REGION Network 5: DataIn - Sollevatori
   RUNG wire#powerrail
      "ValveMachine_PB_Connector"(Enable := TRUE, HMI_PB := "A03_HMI".MB3.Button.A0301.P2.Sollevatori, LB_PB_Rest := FALSE, LB_PB_Work := FALSE, LB_PB_StartStop := FALSE, Other_PB := "A03_HMI".MB3.Button.PB_Empty.Valve, PB => "A0301_Fermi_P2".Sollevatori[1].DataIn.PB)
   END_RUNG
   // the same network as SCL:
   "ValveMachine_PB_Connector"(Enable := TRUE,
                           HMI_PB := "A03_HMI".MB3.Button.A0301.P2.Sollevatori,
                           LB_PB_Rest := FALSE,
                           LB_PB_Work := FALSE,
                           LB_PB_StartStop := FALSE,
                           Other_PB := "A03_HMI".MB3.Button.PB_Empty.Valve,
                           PB => "A0301_Fermi_P2".Sollevatori[1].DataIn.PB);
END_REGION

REGION Network 6 (SCL): DataIn - Sollevatori [1..6]
   // TRASFERIMENTO STATO PULSANTI - Comando manuale diretto 
   "A0301_Fermi_P2".Sollevatori[6].DataIn.PB := "A0301_Fermi_P2".Sollevatori[5].DataIn.PB := "A0301_Fermi_P2".Sollevatori[4].DataIn.PB :=
   "A0301_Fermi_P2".Sollevatori[3].DataIn.PB := "A0301_Fermi_P2".Sollevatori[2].DataIn.PB := "A0301_Fermi_P2".Sollevatori[1].DataIn.PB;
END_REGION

REGION Network 7: << RICHIAMO STAZIONE 2 - FERMI P2 >>
   RUNG wire#powerrail
      "A0301_Fermi_P2"(AreaInterface := "Area03".AreaInterface, ZSI := "F_DB".ZSI_Zone21, DSI := "F_DB".DSI_V_Air_A0301_A0302, DataIn :=, CIn :=, Config := "PrjConfig_A03".A0301.Fermi_P2, MachineInterface =>, COut =>)
   END_RUNG
   // the same network as SCL:
   "A0301_Fermi_P2"(AreaInterface := "Area03".AreaInterface,   // "A0301_Fermi_P2_FB"
                    ZSI := "F_DB".ZSI_Zone21,
                    DSI := "F_DB".DSI_V_Air_A0301_A0302,
                    Config := "PrjConfig_A03".A0301.Fermi_P2);
END_REGION

REGION Network 8 (SCL): << TRASFERIMENTO stati DataOut >>
   REGION COMANDO DELLE USCITE FERMI P2

       // Fermi blocco prodotto Stazione P2 - RIPOSO
       // 
       "A0301_CinghiaTrasporto_1.1_V_Rest_7" := "A0301_Fermi_P2".Fermi[1].DataOut.RestSolenoid;
       "A0301_CinghiaTrasporto_2.1_V_Rest_7" := "A0301_Fermi_P2".Fermi[2].DataOut.RestSolenoid;
       "A0301_CinghiaTrasporto_3.1_V_Rest_7" := "A0301_Fermi_P2".Fermi[3].DataOut.RestSolenoid;
       "A0301_CinghiaTrasporto_4.1_V_Rest_7" := "A0301_Fermi_P2".Fermi[4].DataOut.RestSolenoid;
       "A0301_CinghiaTrasporto_5.1_V_Rest_7" := "A0301_Fermi_P2".Fermi[5].DataOut.RestSolenoid;
       "A0301_CinghiaTrasporto_6.1_V_Rest_7" := "A0301_Fermi_P2".Fermi[6].DataOut.RestSolenoid;

       // Fermi blocco prodotto Stazione P2 - LAVORO
       // 
       "A0301_CinghiaTrasporto_1.1_V_Work_8" := "A0301_Fermi_P2".Fermi[1].DataOut.WorkSolenoid;
       "A0301_CinghiaTrasporto_2.1_V_Work_8" := "A0301_Fermi_P2".Fermi[2].DataOut.WorkSolenoid;
       "A0301_CinghiaTrasporto_3.1_V_Work_8" := "A0301_Fermi_P2".Fermi[3].DataOut.WorkSolenoid;
       "A0301_CinghiaTrasporto_4.1_V_Work_8" := "A0301_Fermi_P2".Fermi[4].DataOut.WorkSolenoid;
       "A0301_CinghiaTrasporto_5.1_V_Work_8" := "A0301_Fermi_P2".Fermi[5].DataOut.WorkSolenoid;
       "A0301_CinghiaTrasporto_6.1_V_Work_8" := "A0301_Fermi_P2".Fermi[6].DataOut.WorkSolenoid;
   END_REGION ;

   REGION COMANDO DELLE USCITE SOLLEVATORE P2
       // Sollevatore Semi guscio prodotto Stazione P2 - RIPOSO
       // 
       "A0301_CinghiaTrasporto_1.1_V_Rest_5" := "A0301_Fermi_P2".Sollevatori[1].DataOut.RestSolenoid;
       "A0301_CinghiaTrasporto_2.1_V_Rest_5" := "A0301_Fermi_P2".Sollevatori[2].DataOut.RestSolenoid;
       "A0301_CinghiaTrasporto_3.1_V_Rest_5" := "A0301_Fermi_P2".Sollevatori[3].DataOut.RestSolenoid;
       "A0301_CinghiaTrasporto_4.1_V_Rest_5" := "A0301_Fermi_P2".Sollevatori[4].DataOut.RestSolenoid;
       "A0301_CinghiaTrasporto_5.1_V_Rest_5" := "A0301_Fermi_P2".Sollevatori[5].DataOut.RestSolenoid;
       "A0301_CinghiaTrasporto_6.1_V_Rest_5" := "A0301_Fermi_P2".Sollevatori[6].DataOut.RestSolenoid;

       // Sollevatore Semi guscio prodotto Stazione P2 - LAVORO
       // 
       "A0301_CinghiaTrasporto_1.1_V_Work_6" := "A0301_Fermi_P2".Sollevatori[1].DataOut.WorkSolenoid;
       "A0301_CinghiaTrasporto_2.1_V_Work_6" := "A0301_Fermi_P2".Sollevatori[2].DataOut.WorkSolenoid;
       "A0301_CinghiaTrasporto_3.1_V_Work_6" := "A0301_Fermi_P2".Sollevatori[3].DataOut.WorkSolenoid;
       "A0301_CinghiaTrasporto_4.1_V_Work_6" := "A0301_Fermi_P2".Sollevatori[4].DataOut.WorkSolenoid;
       "A0301_CinghiaTrasporto_5.1_V_Work_6" := "A0301_Fermi_P2".Sollevatori[5].DataOut.WorkSolenoid;
       "A0301_CinghiaTrasporto_6.1_V_Work_6" := "A0301_Fermi_P2".Sollevatori[6].DataOut.WorkSolenoid;

   END_REGION ;*)
END_REGION
END_FUNCTION

FUNCTION_BLOCK "A0301_Fermi_P2_FB"   // FB62, LAD
TITLE = == GESTIONE DELLA STAZIONE P2 ==
// stored: MemoryReserve 100, SetENOAutomatically false
   VAR_INPUT
      AreaInterface : "AreaInterface";
      ZSI : "udt_ZoneSafetyInterface";
      DSI : "udt_DeviceSafetyInterface";
      DataIn : Struct
         OP_Rest_PB : Bool;
         OP_Work_PB : Bool;
      END_STRUCT;
      CIn : Struct
         Manager_Fermi : "ValveMachine_Manager";
         Manager_Sollevatori : "ValveMachine_Manager";
         SemiAut : Bool;
         P1 : Struct
            Fermi : "ValveMachine_COut";
            Pareggiatore : "ValveMachine_COut";
         END_STRUCT;
         Trasporto : "SpeedMachine_COut";
         Sts_Ribalta : Struct
            Pos0_Reached : Bool;
            Pos1_Reached : Bool;
            Pos2_Reached : Bool;
            Pos3_Reached : Bool;
         END_STRUCT;
      END_STRUCT;
      Config : Struct
         Fermi : Array[1..6] of "ValveMachine_Config";
         Sollevatori : Array[1..6] of "ValveMachine_Config";
         DelayMissingCondition : Time := T#3s;
      END_STRUCT;
   END_VAR
   VAR_OUTPUT
      MachineInterface : "MachineInterface";
      COut : Struct
         Fermi : "ValveMachine_COut";
         Sollevatori : "ValveMachine_COut";
      END_STRUCT;
   END_VAR
   VAR
      Alarm : Struct
         Fermi : Array[1..6] of "ValveAlr";
         Sollevatori { S7_SetPoint := 'True'} : Array[1..6] of "ValveAlr";
      END_STRUCT;
      Warning : Struct
         OP_REST_MissingCnd : Bool;   // Mancanza comando arresto
         OP_WORK_MissingCnd : Bool;   // Mancanza consenso lavoro
         Fermi : Array[1..6] of "ValveMachine_Wng";
         Sollevatori { S7_SetPoint := 'True'} : Array[1..6] of "ValveMachine_Wng";
      END_STRUCT;
      HMI : Struct
         Selection : Array[1..6] of Bool;   // 0=Disable / 1=Enable Pin
         FermiSts { S7_SetPoint := 'True'} : "UDT_HMI-Sts_ValvePosA0301";
         SollevatoriSts { S7_SetPoint := 'True'} : "UDT_HMI-Sts_ValvePosA0301";
      END_STRUCT;
      Sts : Struct
         Fermi_AlarmPresence : Bool;
         Sollevatori_AlarmPresence : Bool;
         OP_CanMoveFreely : Bool;
         OP_Rest_Cnd : Bool;
         Op_Work_Cnd : Bool;
      END_STRUCT;
      Ctrl : Struct
         OP_Rest_Man : Bool;
         OP_Work_Man : Bool;
         OP_Rest_Aut : Bool;
         OP_Work_Aut : Bool;
         OP_Rest : Bool;
         OP_Work : Bool;
      END_STRUCT;
      Fermi : Array[1..6] of "ValveMachine_FB";
      Sollevatori { S7_SetPoint := 'True'} : Array[1..6] of "ValveMachine_FB";
      AUX : Struct
         OP_Rest_PB : Bool;
         OP_Work_PB : Bool;
      END_STRUCT;
      TON_OP_REST_MissingCnd { S7_SetPoint := 'True'} : TON_TIME;
      TON_OP_WORK_MissingCnd { S7_SetPoint := 'True'} : TON_TIME;
      TON_Anticipi : Struct
         Rest : Struct
            Sollevatori { S7_SetPoint := 'True'} : IEC_TIMER;
         END_STRUCT;
         Work : Struct
            Sollevatori : IEC_TIMER;
         END_STRUCT;
      END_STRUCT;
   END_VAR
   VAR_TEMP
      PE : Struct
         OP_Rest_PB : Bool;
         OP_Work_PB : Bool;
      END_STRUCT;
      Anticipi : Struct
         Sollevatori : Struct
            COut_Work : Bool;
            COut_Rest : Bool;
            Not_Ls_Work : Bool;
            Not_Ls_Rest : Bool;
         END_STRUCT;
      END_STRUCT;
   END_VAR
   VAR_TEMP   // added for the SCL form of the ladder/FBD networks
      _w1 : Bool;
      _w2 : Bool;
      _w3 : Bool;
      _w4 : Bool;
   END_VAR
BEGIN

REGION Network 2: Anticipi Movimento LAVORO
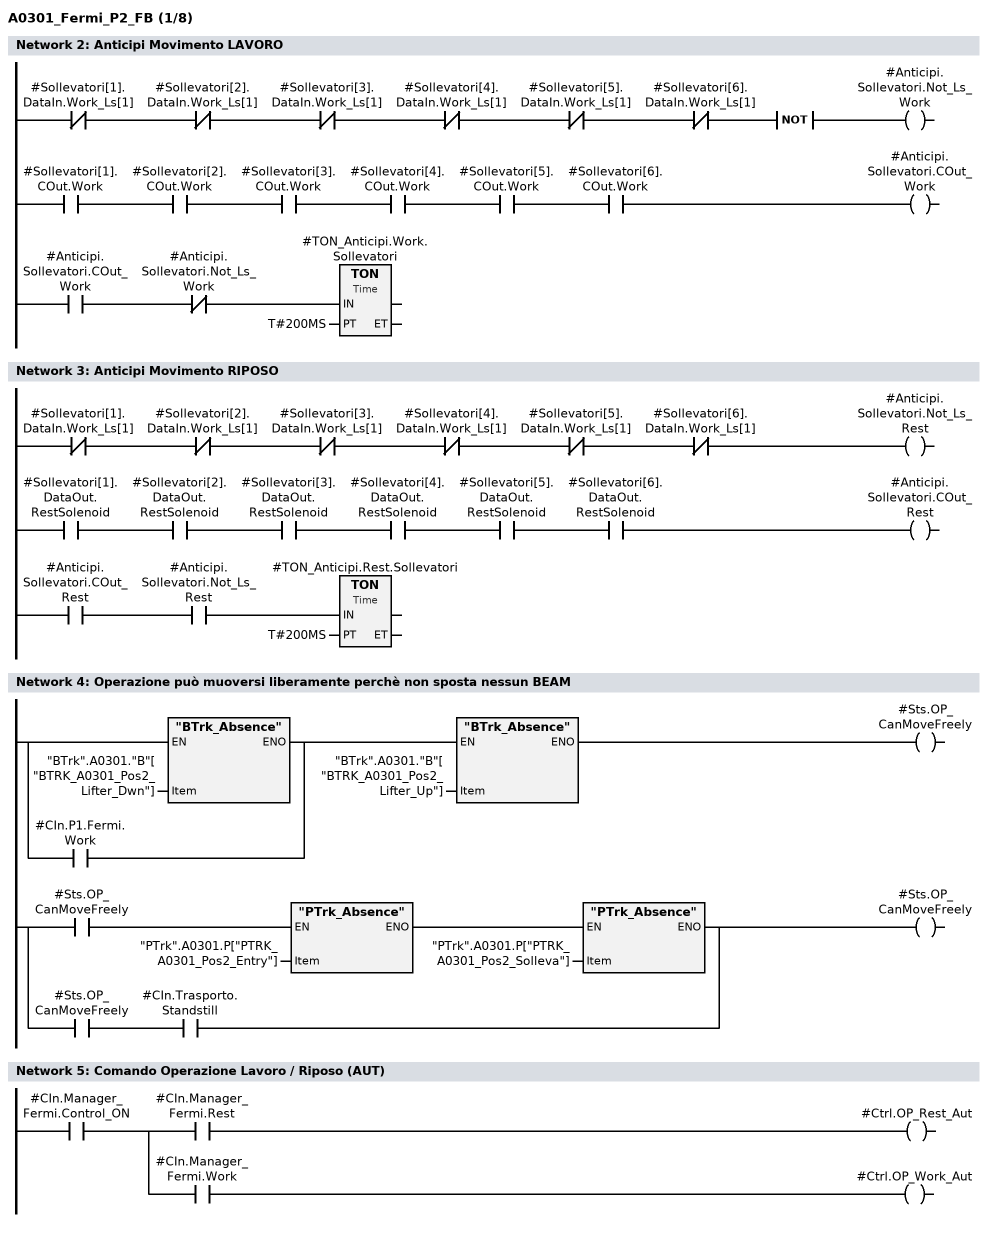
   RUNG wire#powerrail
      I_Contact( #Sollevatori[1].DataIn.Work_Ls[1] )
      I_Contact( #Sollevatori[2].DataIn.Work_Ls[1] )
      I_Contact( #Sollevatori[3].DataIn.Work_Ls[1] )
      I_Contact( #Sollevatori[4].DataIn.Work_Ls[1] )
      I_Contact( #Sollevatori[5].DataIn.Work_Ls[1] )
      I_Contact( #Sollevatori[6].DataIn.Work_Ls[1] )
      Not()
      Coil( #Anticipi.Sollevatori.Not_Ls_Work )
   END_RUNG
   RUNG wire#powerrail
      Contact( #Sollevatori[1].COut.Work )
      Contact( #Sollevatori[2].COut.Work )
      Contact( #Sollevatori[3].COut.Work )
      Contact( #Sollevatori[4].COut.Work )
      Contact( #Sollevatori[5].COut.Work )
      Contact( #Sollevatori[6].COut.Work )
      Coil( #Anticipi.Sollevatori.COut_Work )
   END_RUNG
   RUNG wire#powerrail
      Contact( #Anticipi.Sollevatori.COut_Work )
      I_Contact( #Anticipi.Sollevatori.Not_Ls_Work )
      { S7_Templates := "time_type := Time" } #TON_Anticipi.Work.Sollevatori.TON(pt := T#200MS, et =>)
   END_RUNG
   // the same network as SCL:
   #Anticipi.Sollevatori.Not_Ls_Work := NOT (NOT #Sollevatori[1].DataIn.Work_Ls[1] AND NOT #Sollevatori[2].DataIn.Work_Ls[1] AND NOT #Sollevatori[3].DataIn.Work_Ls[1] AND NOT #Sollevatori[4].DataIn.Work_Ls[1] AND NOT #Sollevatori[5].DataIn.Work_Ls[1] AND NOT #Sollevatori[6].DataIn.Work_Ls[1]);
   #Anticipi.Sollevatori.COut_Work := #Sollevatori[1].COut.Work AND #Sollevatori[2].COut.Work AND #Sollevatori[3].COut.Work AND #Sollevatori[4].COut.Work AND #Sollevatori[5].COut.Work AND #Sollevatori[6].COut.Work;
   #TON_Anticipi.Work.Sollevatori.TON(IN := #Anticipi.Sollevatori.COut_Work AND NOT #Anticipi.Sollevatori.Not_Ls_Work,
                           PT := T#200MS);
END_REGION

REGION Network 3: Anticipi Movimento RIPOSO
   RUNG wire#powerrail
      I_Contact( #Sollevatori[1].DataIn.Work_Ls[1] )
      I_Contact( #Sollevatori[2].DataIn.Work_Ls[1] )
      I_Contact( #Sollevatori[3].DataIn.Work_Ls[1] )
      I_Contact( #Sollevatori[4].DataIn.Work_Ls[1] )
      I_Contact( #Sollevatori[5].DataIn.Work_Ls[1] )
      I_Contact( #Sollevatori[6].DataIn.Work_Ls[1] )
      Coil( #Anticipi.Sollevatori.Not_Ls_Rest )
   END_RUNG
   RUNG wire#powerrail
      Contact( #Sollevatori[1].DataOut.RestSolenoid )
      Contact( #Sollevatori[2].DataOut.RestSolenoid )
      Contact( #Sollevatori[3].DataOut.RestSolenoid )
      Contact( #Sollevatori[4].DataOut.RestSolenoid )
      Contact( #Sollevatori[5].DataOut.RestSolenoid )
      Contact( #Sollevatori[6].DataOut.RestSolenoid )
      Coil( #Anticipi.Sollevatori.COut_Rest )
   END_RUNG
   RUNG wire#powerrail
      Contact( #Anticipi.Sollevatori.COut_Rest )
      Contact( #Anticipi.Sollevatori.Not_Ls_Rest )
      { S7_Templates := "time_type := Time" } #TON_Anticipi.Rest.Sollevatori.TON(pt := T#200MS, et =>)
   END_RUNG
   // the same network as SCL:
   #Anticipi.Sollevatori.Not_Ls_Rest := NOT #Sollevatori[1].DataIn.Work_Ls[1] AND NOT #Sollevatori[2].DataIn.Work_Ls[1] AND NOT #Sollevatori[3].DataIn.Work_Ls[1] AND NOT #Sollevatori[4].DataIn.Work_Ls[1] AND NOT #Sollevatori[5].DataIn.Work_Ls[1] AND NOT #Sollevatori[6].DataIn.Work_Ls[1];
   #Anticipi.Sollevatori.COut_Rest := #Sollevatori[1].DataOut.RestSolenoid AND #Sollevatori[2].DataOut.RestSolenoid AND #Sollevatori[3].DataOut.RestSolenoid AND #Sollevatori[4].DataOut.RestSolenoid AND #Sollevatori[5].DataOut.RestSolenoid AND #Sollevatori[6].DataOut.RestSolenoid;
   #TON_Anticipi.Rest.Sollevatori.TON(IN := #Anticipi.Sollevatori.COut_Rest AND #Anticipi.Sollevatori.Not_Ls_Rest,
                           PT := T#200MS);
END_REGION

REGION Network 4: Operazione può muoversi liberamente perchè non sposta nessun BEAM
   RUNG wire#powerrail
      "BTrk_Absence"(Item := "BTrk".A0301."B"["BTRK_A0301_Pos2_Lifter_Dwn"])
      wire#w1
      "BTrk_Absence"(Item := "BTrk".A0301."B"["BTRK_A0301_Pos2_Lifter_Up"])
      Coil( #Sts.OP_CanMoveFreely )
   END_RUNG
   RUNG wire#powerrail
      Contact( #CIn.P1.Fermi.Work )
   END_RUNG wire#w1
   RUNG wire#powerrail
      Contact( #Sts.OP_CanMoveFreely )
      "PTrk_Absence"(Item := "PTrk".A0301.P["PTRK_A0301_Pos2_Entry"])
      "PTrk_Absence"(Item := "PTrk".A0301.P["PTRK_A0301_Pos2_Solleva"])
      wire#w2
      Coil( #Sts.OP_CanMoveFreely )
   END_RUNG
   RUNG wire#powerrail
      Contact( #Sts.OP_CanMoveFreely )
      Contact( #CIn.Trasporto.Standstill )
   END_RUNG wire#w2
   // the same network as SCL:
   "BTrk_Absence"(Item := "BTrk".A0301."B"["BTRK_A0301_Pos2_Lifter_Dwn"], ENO => #_w1);
   "BTrk_Absence"(EN := #_w1 OR #CIn.P1.Fermi.Work,
                  Item := "BTrk".A0301."B"["BTRK_A0301_Pos2_Lifter_Up"],
                  ENO => #_w2);
   #Sts.OP_CanMoveFreely := #_w2;
   "PTrk_Absence"(EN := #Sts.OP_CanMoveFreely, Item := "PTrk".A0301.P["PTRK_A0301_Pos2_Entry"], ENO => #_w3);
   "PTrk_Absence"(EN := #_w3, Item := "PTrk".A0301.P["PTRK_A0301_Pos2_Solleva"], ENO => #_w4);
   #Sts.OP_CanMoveFreely := #_w4 OR (#Sts.OP_CanMoveFreely AND #CIn.Trasporto.Standstill);
END_REGION

REGION Network 5: Comando Operazione Lavoro / Riposo (AUT)
   RUNG wire#powerrail
      Contact( #CIn.Manager_Fermi.Control_ON )
      wire#w1
      Contact( #CIn.Manager_Fermi.Rest )
      Coil( #Ctrl.OP_Rest_Aut )
   END_RUNG
   RUNG wire#w1
      Contact( #CIn.Manager_Fermi.Work )
      Coil( #Ctrl.OP_Work_Aut )
   END_RUNG
   // the same network as SCL:
   #Ctrl.OP_Rest_Aut := #CIn.Manager_Fermi.Control_ON AND #CIn.Manager_Fermi.Rest;
   #Ctrl.OP_Work_Aut := #CIn.Manager_Fermi.Control_ON AND #CIn.Manager_Fermi.Work;
END_REGION

REGION Network 6: Comando Operazione Lavoro / Riposo (MAN)
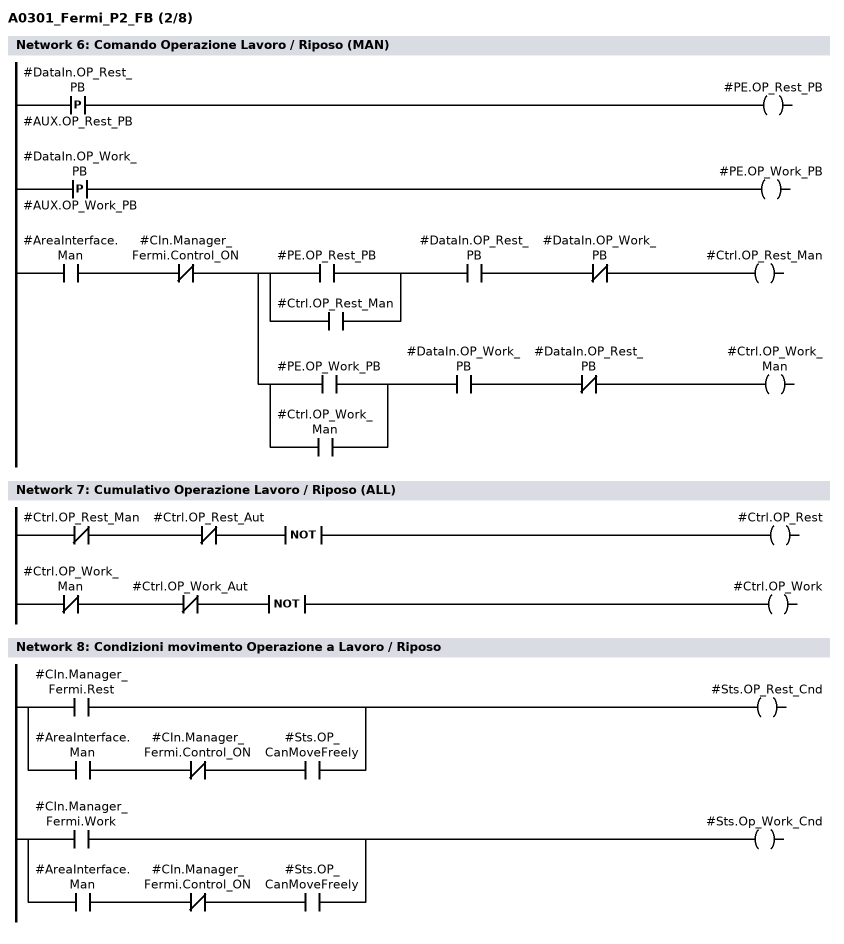
   RUNG wire#powerrail
      P_Contact(operand := #DataIn.OP_Rest_PB, bit := #AUX.OP_Rest_PB)
      Coil( #PE.OP_Rest_PB )
   END_RUNG
   RUNG wire#powerrail
      P_Contact(operand := #DataIn.OP_Work_PB, bit := #AUX.OP_Work_PB)
      Coil( #PE.OP_Work_PB )
   END_RUNG
   RUNG wire#powerrail
      Contact( #AreaInterface.Man )
      I_Contact( #CIn.Manager_Fermi.Control_ON )
      wire#w1
      Contact( #PE.OP_Rest_PB )
      wire#w2
      Contact( #DataIn.OP_Rest_PB )
      I_Contact( #DataIn.OP_Work_PB )
      Coil( #Ctrl.OP_Rest_Man )
   END_RUNG
   RUNG wire#w1
      Contact( #Ctrl.OP_Rest_Man )
   END_RUNG wire#w2
   RUNG wire#w1
      Contact( #PE.OP_Work_PB )
      wire#w3
      Contact( #DataIn.OP_Work_PB )
      I_Contact( #DataIn.OP_Rest_PB )
      Coil( #Ctrl.OP_Work_Man )
   END_RUNG
   RUNG wire#w1
      Contact( #Ctrl.OP_Work_Man )
   END_RUNG wire#w3
   // the same network as SCL:
   #_w1 := #DataIn.OP_Rest_PB AND NOT #AUX.OP_Rest_PB;   // rising edge of #DataIn.OP_Rest_PB
   #AUX.OP_Rest_PB := #DataIn.OP_Rest_PB;
   #PE.OP_Rest_PB := #_w1;
   #_w2 := #DataIn.OP_Work_PB AND NOT #AUX.OP_Work_PB;   // rising edge of #DataIn.OP_Work_PB
   #AUX.OP_Work_PB := #DataIn.OP_Work_PB;
   #PE.OP_Work_PB := #_w2;
   #_w3 := #AreaInterface.Man AND NOT #CIn.Manager_Fermi.Control_ON;
   #Ctrl.OP_Rest_Man := #_w3 AND (#PE.OP_Rest_PB OR #Ctrl.OP_Rest_Man) AND #DataIn.OP_Rest_PB AND NOT #DataIn.OP_Work_PB;
   #Ctrl.OP_Work_Man := #_w3 AND (#PE.OP_Work_PB OR #Ctrl.OP_Work_Man) AND #DataIn.OP_Work_PB AND NOT #DataIn.OP_Rest_PB;
END_REGION

REGION Network 7: Cumulativo Operazione Lavoro / Riposo (ALL)
   RUNG wire#powerrail
      I_Contact( #Ctrl.OP_Rest_Man )
      I_Contact( #Ctrl.OP_Rest_Aut )
      Not()
      Coil( #Ctrl.OP_Rest )
   END_RUNG
   RUNG wire#powerrail
      I_Contact( #Ctrl.OP_Work_Man )
      I_Contact( #Ctrl.OP_Work_Aut )
      Not()
      Coil( #Ctrl.OP_Work )
   END_RUNG
   // the same network as SCL:
   #Ctrl.OP_Rest := NOT (NOT #Ctrl.OP_Rest_Man AND NOT #Ctrl.OP_Rest_Aut);
   #Ctrl.OP_Work := NOT (NOT #Ctrl.OP_Work_Man AND NOT #Ctrl.OP_Work_Aut);
END_REGION

REGION Network 8: Condizioni movimento Operazione a Lavoro / Riposo
   RUNG wire#powerrail
      Contact( #CIn.Manager_Fermi.Rest )
      wire#w1
      Coil( #Sts.OP_Rest_Cnd )
   END_RUNG
   RUNG wire#powerrail
      Contact( #AreaInterface.Man )
      I_Contact( #CIn.Manager_Fermi.Control_ON )
      Contact( #Sts.OP_CanMoveFreely )
   END_RUNG wire#w1
   RUNG wire#powerrail
      Contact( #CIn.Manager_Fermi.Work )
      wire#w2
      Coil( #Sts.Op_Work_Cnd )
   END_RUNG
   RUNG wire#powerrail
      Contact( #AreaInterface.Man )
      I_Contact( #CIn.Manager_Fermi.Control_ON )
      Contact( #Sts.OP_CanMoveFreely )
   END_RUNG wire#w2
   // the same network as SCL:
   #Sts.OP_Rest_Cnd := #CIn.Manager_Fermi.Rest OR (#AreaInterface.Man AND NOT #CIn.Manager_Fermi.Control_ON AND #Sts.OP_CanMoveFreely);
   #Sts.Op_Work_Cnd := #CIn.Manager_Fermi.Work OR (#AreaInterface.Man AND NOT #CIn.Manager_Fermi.Control_ON AND #Sts.OP_CanMoveFreely);
END_REGION

REGION Network 10 (SCL): Fermi + Sollevatore - Cin Manager (Esecuzione sequenza comandi)
   //
   #Fermi[1].Cin.Manager.Rest := FALSE;
   #Fermi[2].Cin.Manager.Rest := FALSE;
   #Fermi[3].Cin.Manager.Rest := FALSE;
   #Fermi[4].Cin.Manager.Rest := FALSE;
   #Fermi[5].Cin.Manager.Rest := FALSE;
   #Fermi[6].Cin.Manager.Rest := FALSE;
   #Sollevatori[1].Cin.Manager.Rest := FALSE;
   #Sollevatori[2].Cin.Manager.Rest := FALSE;
   #Sollevatori[3].Cin.Manager.Rest := FALSE;
   #Sollevatori[4].Cin.Manager.Rest := FALSE;
   #Sollevatori[5].Cin.Manager.Rest := FALSE;
   #Sollevatori[6].Cin.Manager.Rest := FALSE;


   //************************************
   #Fermi[1].Cin.Manager.Work := FALSE;
   #Fermi[2].Cin.Manager.Work := FALSE;
   #Fermi[3].Cin.Manager.Work := FALSE;
   #Fermi[4].Cin.Manager.Work := FALSE;
   #Fermi[5].Cin.Manager.Work := FALSE;
   #Fermi[6].Cin.Manager.Work := FALSE;
   #Sollevatori[1].Cin.Manager.Work := FALSE;
   #Sollevatori[2].Cin.Manager.Work := FALSE;
   #Sollevatori[3].Cin.Manager.Work := FALSE;
   #Sollevatori[4].Cin.Manager.Work := FALSE;
   #Sollevatori[5].Cin.Manager.Work := FALSE;
   #Sollevatori[6].Cin.Manager.Work := FALSE;
   //
   // CIn Manager  Control ON se ho un richiesta di comando attiva
   IF #AreaInterface.Aut OR #CIn.SemiAut THEN
       #Fermi[1].Cin.Manager.Control_ON := TRUE;
       #Fermi[2].Cin.Manager.Control_ON := TRUE;
       #Fermi[3].Cin.Manager.Control_ON := TRUE;
       #Fermi[4].Cin.Manager.Control_ON := TRUE;
       #Fermi[5].Cin.Manager.Control_ON := TRUE;
       #Fermi[6].Cin.Manager.Control_ON := TRUE;
       #Sollevatori[1].Cin.Manager.Control_ON := TRUE;
       #Sollevatori[2].Cin.Manager.Control_ON := TRUE;
       #Sollevatori[3].Cin.Manager.Control_ON := TRUE;
       #Sollevatori[4].Cin.Manager.Control_ON := TRUE;
       #Sollevatori[5].Cin.Manager.Control_ON := TRUE;
       #Sollevatori[6].Cin.Manager.Control_ON := TRUE;
   ELSE
       #Fermi[1].Cin.Manager.Control_ON := FALSE;
       #Fermi[2].Cin.Manager.Control_ON := FALSE;
       #Fermi[3].Cin.Manager.Control_ON := FALSE;
       #Fermi[4].Cin.Manager.Control_ON := FALSE;
       #Fermi[5].Cin.Manager.Control_ON := FALSE;
       #Fermi[6].Cin.Manager.Control_ON := FALSE;
       #Sollevatori[1].Cin.Manager.Control_ON := FALSE;
       #Sollevatori[2].Cin.Manager.Control_ON := FALSE;
       #Sollevatori[3].Cin.Manager.Control_ON := FALSE;
       #Sollevatori[4].Cin.Manager.Control_ON := FALSE;
       #Sollevatori[5].Cin.Manager.Control_ON := FALSE;
       #Sollevatori[6].Cin.Manager.Control_ON := FALSE;
   END_IF;

   // Comando CIn Manager Work FERMI
   IF #Ctrl.OP_Work_Aut AND #Sts.Op_Work_Cnd AND #COut.Sollevatori.Rest THEN

       #Fermi[1].Cin.Manager.Work := TRUE;
       #Fermi[2].Cin.Manager.Work := TRUE;
       #Fermi[3].Cin.Manager.Work := TRUE;
       #Fermi[4].Cin.Manager.Work := TRUE;
       #Fermi[5].Cin.Manager.Work := TRUE;
       #Fermi[6].Cin.Manager.Work := TRUE;

   END_IF;

   // Comando CIn Manager Work SOLLEVATORE se fermi sono alti
   IF #CIn.Manager_Sollevatori.Work THEN
       #Sollevatori[1].Cin.Manager.Work := TRUE;
       #Sollevatori[2].Cin.Manager.Work := TRUE;
       #Sollevatori[3].Cin.Manager.Work := TRUE;
       #Sollevatori[4].Cin.Manager.Work := TRUE;
       #Sollevatori[5].Cin.Manager.Work := TRUE;
       #Sollevatori[6].Cin.Manager.Work := TRUE;
   END_IF;


   // Comando CIn Manager Rest FERMI se Sollevatore è basso
   IF #Ctrl.OP_Rest_Aut AND #Sts.OP_Rest_Cnd AND NOT #Ctrl.OP_Work_Aut AND #COut.Sollevatori.Rest THEN

       #Fermi[1].Cin.Manager.Rest := TRUE;
       #Fermi[2].Cin.Manager.Rest := TRUE;
       #Fermi[3].Cin.Manager.Rest := TRUE;
       #Fermi[4].Cin.Manager.Rest := TRUE;
       #Fermi[5].Cin.Manager.Rest := TRUE;
       #Fermi[6].Cin.Manager.Rest := TRUE;

       // Quando il sollevatore è alto i fermi scendono
   ELSIF #COut.Sollevatori.Work THEN
       #Fermi[1].Cin.Manager.Rest := TRUE;
       #Fermi[2].Cin.Manager.Rest := TRUE;
       #Fermi[3].Cin.Manager.Rest := TRUE;
       #Fermi[4].Cin.Manager.Rest := TRUE;
       #Fermi[5].Cin.Manager.Rest := TRUE;
       #Fermi[6].Cin.Manager.Rest := TRUE;

   END_IF;

    //Quando i sollevatori sono alti e i fermi bassi e ho comando arresto abbasso abbasso i Sollevatori
   IF #CIn.Manager_Sollevatori.Rest THEN
       #Sollevatori[1].Cin.Manager.Rest := TRUE;
       #Sollevatori[2].Cin.Manager.Rest := TRUE;
       #Sollevatori[3].Cin.Manager.Rest := TRUE;
       #Sollevatori[4].Cin.Manager.Rest := TRUE;
       #Sollevatori[5].Cin.Manager.Rest := TRUE;
       #Sollevatori[6].Cin.Manager.Rest := TRUE;
   END_IF;
END_REGION

REGION Network 11 (SCL): CIn Abilitazioni Stop Manager
   //
   // CIn Manager Stop per richiesta apertura safety
   IF #CIn.Manager_Fermi.EnableStopDoorOpeningReq THEN
       #Fermi[1].Cin.Manager.EnableStopDoorOpeningReq := TRUE;
       #Fermi[2].Cin.Manager.EnableStopDoorOpeningReq := TRUE;
       #Fermi[3].Cin.Manager.EnableStopDoorOpeningReq := TRUE;
       #Fermi[4].Cin.Manager.EnableStopDoorOpeningReq := TRUE;
       #Fermi[5].Cin.Manager.EnableStopDoorOpeningReq := TRUE;
       #Fermi[6].Cin.Manager.EnableStopDoorOpeningReq := TRUE;
       #Sollevatori[1].Cin.Manager.EnableStopDoorOpeningReq := TRUE;
       #Sollevatori[2].Cin.Manager.EnableStopDoorOpeningReq := TRUE;
       #Sollevatori[3].Cin.Manager.EnableStopDoorOpeningReq := TRUE;
       #Sollevatori[4].Cin.Manager.EnableStopDoorOpeningReq := TRUE;
       #Sollevatori[5].Cin.Manager.EnableStopDoorOpeningReq := TRUE;
       #Sollevatori[6].Cin.Manager.EnableStopDoorOpeningReq := TRUE;
   ELSE
       #Fermi[1].Cin.Manager.EnableStopDoorOpeningReq := FALSE;
       #Fermi[2].Cin.Manager.EnableStopDoorOpeningReq := FALSE;
       #Fermi[3].Cin.Manager.EnableStopDoorOpeningReq := FALSE;
       #Fermi[4].Cin.Manager.EnableStopDoorOpeningReq := FALSE;
       #Fermi[5].Cin.Manager.EnableStopDoorOpeningReq := FALSE;
       #Fermi[6].Cin.Manager.EnableStopDoorOpeningReq := FALSE;
       #Sollevatori[1].Cin.Manager.EnableStopDoorOpeningReq := FALSE;
       #Sollevatori[2].Cin.Manager.EnableStopDoorOpeningReq := FALSE;
       #Sollevatori[3].Cin.Manager.EnableStopDoorOpeningReq := FALSE;
       #Sollevatori[4].Cin.Manager.EnableStopDoorOpeningReq := FALSE;
       #Sollevatori[5].Cin.Manager.EnableStopDoorOpeningReq := FALSE;
       #Sollevatori[6].Cin.Manager.EnableStopDoorOpeningReq := FALSE;

   END_IF;
   // CIn Manager Stop in fase delle macchine precedenti
   IF #CIn.Manager_Fermi.EnableStopInPhase THEN
       #Fermi[1].Cin.Manager.EnableStopInPhase := TRUE;
       #Fermi[2].Cin.Manager.EnableStopInPhase := TRUE;
       #Fermi[3].Cin.Manager.EnableStopInPhase := TRUE;
       #Fermi[4].Cin.Manager.EnableStopInPhase := TRUE;
       #Fermi[5].Cin.Manager.EnableStopInPhase := TRUE;
       #Fermi[6].Cin.Manager.EnableStopInPhase := TRUE;
       #Sollevatori[1].Cin.Manager.EnableStopInPhase := TRUE;
       #Sollevatori[2].Cin.Manager.EnableStopInPhase := TRUE;
       #Sollevatori[3].Cin.Manager.EnableStopInPhase := TRUE;
       #Sollevatori[4].Cin.Manager.EnableStopInPhase := TRUE;
       #Sollevatori[5].Cin.Manager.EnableStopInPhase := TRUE; 
       #Sollevatori[6].Cin.Manager.EnableStopInPhase := TRUE;
   ELSE
       #Fermi[1].Cin.Manager.EnableStopInPhase := FALSE;
       #Fermi[2].Cin.Manager.EnableStopInPhase := FALSE;
       #Fermi[3].Cin.Manager.EnableStopInPhase := FALSE;
       #Fermi[4].Cin.Manager.EnableStopInPhase := FALSE;
       #Fermi[5].Cin.Manager.EnableStopInPhase := FALSE;
       #Fermi[6].Cin.Manager.EnableStopInPhase := FALSE;
       #Sollevatori[1].Cin.Manager.EnableStopInPhase := FALSE;
       #Sollevatori[2].Cin.Manager.EnableStopInPhase := FALSE;
       #Sollevatori[3].Cin.Manager.EnableStopInPhase := FALSE;
       #Sollevatori[4].Cin.Manager.EnableStopInPhase := FALSE;
       #Sollevatori[5].Cin.Manager.EnableStopInPhase := FALSE;
       #Sollevatori[6].Cin.Manager.EnableStopInPhase := FALSE;
   END_IF;

   // CIn Manager Stop programmato configurabile a piacere
   IF #CIn.Manager_Fermi.EnableStopProgrammed THEN
       #Fermi[1].Cin.Manager.EnableStopProgrammed := TRUE;
       #Fermi[2].Cin.Manager.EnableStopProgrammed := TRUE;
       #Fermi[3].Cin.Manager.EnableStopProgrammed := TRUE;
       #Fermi[4].Cin.Manager.EnableStopProgrammed := TRUE;
       #Fermi[5].Cin.Manager.EnableStopProgrammed := TRUE;
       #Fermi[6].Cin.Manager.EnableStopProgrammed := TRUE;
       #Sollevatori[1].Cin.Manager.EnableStopProgrammed := TRUE;
       #Sollevatori[2].Cin.Manager.EnableStopProgrammed := TRUE;
       #Sollevatori[3].Cin.Manager.EnableStopProgrammed := TRUE;
       #Sollevatori[4].Cin.Manager.EnableStopProgrammed := TRUE;
       #Sollevatori[5].Cin.Manager.EnableStopProgrammed := TRUE;
       #Sollevatori[6].Cin.Manager.EnableStopProgrammed := TRUE;
   ELSE
       #Fermi[1].Cin.Manager.EnableStopProgrammed := FALSE;
       #Fermi[2].Cin.Manager.EnableStopProgrammed := FALSE;
       #Fermi[3].Cin.Manager.EnableStopProgrammed := FALSE;
       #Fermi[4].Cin.Manager.EnableStopProgrammed := FALSE;
       #Fermi[5].Cin.Manager.EnableStopProgrammed := FALSE;
       #Fermi[6].Cin.Manager.EnableStopProgrammed := FALSE;
       #Sollevatori[1].Cin.Manager.EnableStopProgrammed := FALSE;
       #Sollevatori[2].Cin.Manager.EnableStopProgrammed := FALSE;
       #Sollevatori[3].Cin.Manager.EnableStopProgrammed := FALSE;
       #Sollevatori[4].Cin.Manager.EnableStopProgrammed := FALSE;
       #Sollevatori[5].Cin.Manager.EnableStopProgrammed := FALSE;
       #Sollevatori[6].Cin.Manager.EnableStopProgrammed := FALSE;
   END_IF;
END_REGION

REGION Network 12: <+>
END_REGION

REGION Network 13: Warning manacanza condizioni esecuzione Operazione RIPOSO / LAVORO
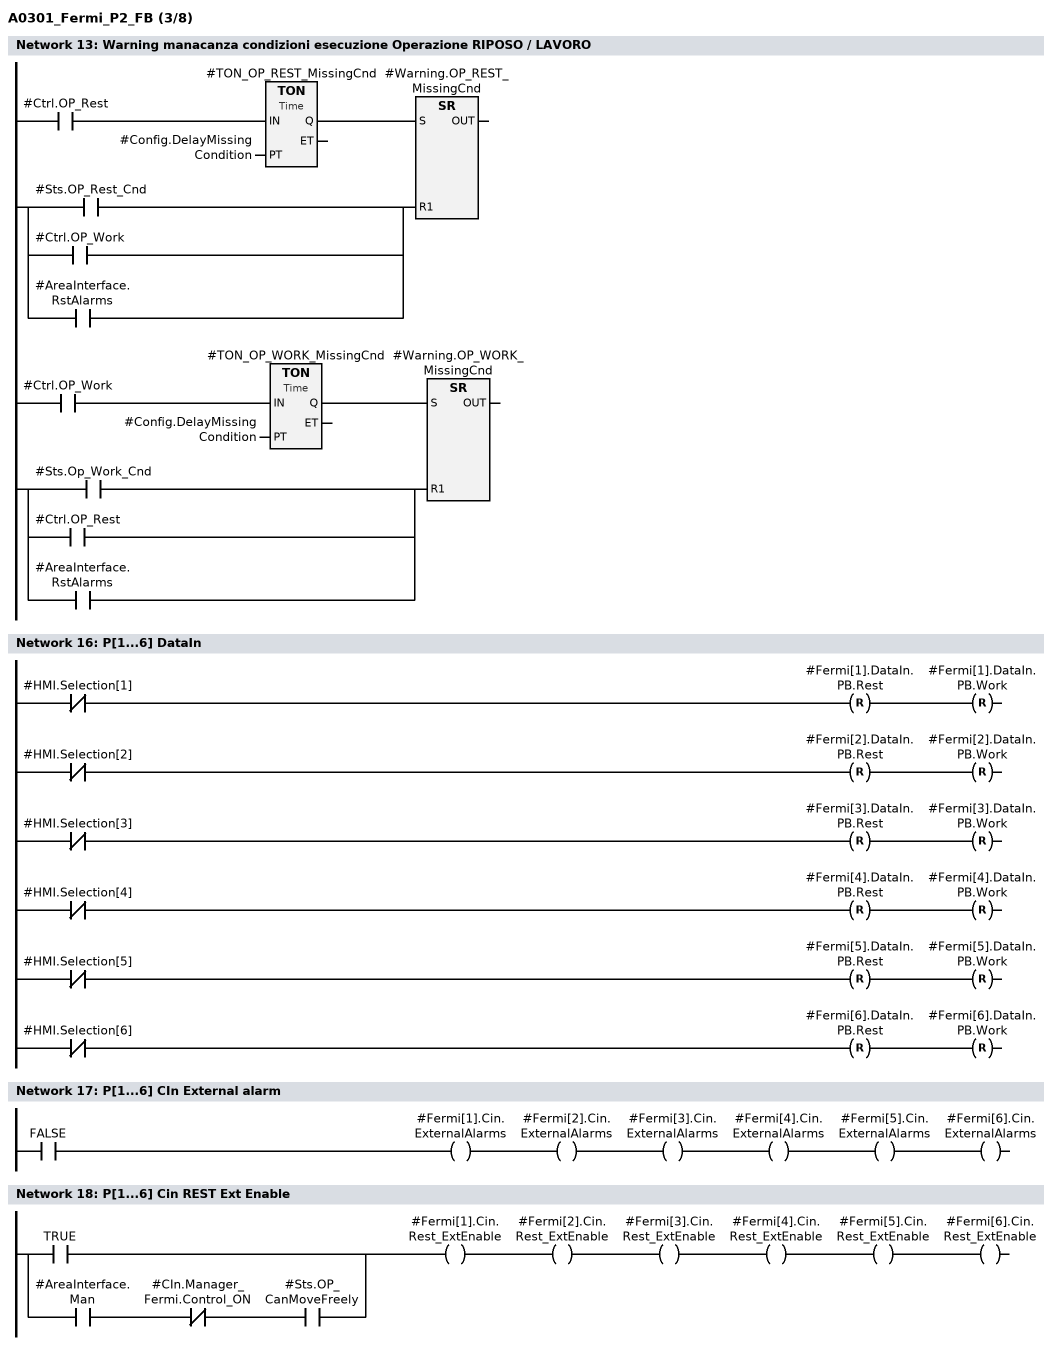
   RUNG wire#powerrail
      Contact( #Ctrl.OP_Rest )
      { S7_Templates := "time_type := Time" } #TON_OP_REST_MissingCnd.TON(pt := #Config.DelayMissingCondition, et =>)
      S_SR(operand := #Warning.OP_REST_MissingCnd, r1 := wire#w1)
   END_RUNG
   RUNG wire#powerrail
      Contact( #Sts.OP_Rest_Cnd )
   END_RUNG wire#w1
   RUNG wire#powerrail
      Contact( #Ctrl.OP_Work )
   END_RUNG wire#w1
   RUNG wire#powerrail
      Contact( #AreaInterface.RstAlarms )
   END_RUNG wire#w1
   RUNG wire#powerrail
      Contact( #Ctrl.OP_Work )
      { S7_Templates := "time_type := Time" } #TON_OP_WORK_MissingCnd.TON(pt := #Config.DelayMissingCondition, et =>)
      S_SR(operand := #Warning.OP_WORK_MissingCnd, r1 := wire#w2)
   END_RUNG
   RUNG wire#powerrail
      Contact( #Sts.Op_Work_Cnd )
   END_RUNG wire#w2
   RUNG wire#powerrail
      Contact( #Ctrl.OP_Rest )
   END_RUNG wire#w2
   RUNG wire#powerrail
      Contact( #AreaInterface.RstAlarms )
   END_RUNG wire#w2
   // the same network as SCL:
   #TON_OP_REST_MissingCnd(IN := #Ctrl.OP_Rest, PT := #Config.DelayMissingCondition);   // TON
   IF #TON_OP_REST_MissingCnd.Q THEN
       #Warning.OP_REST_MissingCnd := TRUE;   // SR flip-flop
   END_IF;
   IF #Sts.OP_Rest_Cnd OR #Ctrl.OP_Work OR #AreaInterface.RstAlarms THEN
       #Warning.OP_REST_MissingCnd := FALSE;
   END_IF;
   #TON_OP_WORK_MissingCnd(IN := #Ctrl.OP_Work, PT := #Config.DelayMissingCondition);   // TON
   IF #TON_OP_WORK_MissingCnd.Q THEN
       #Warning.OP_WORK_MissingCnd := TRUE;   // SR flip-flop
   END_IF;
   IF #Sts.Op_Work_Cnd OR #Ctrl.OP_Rest OR #AreaInterface.RstAlarms THEN
       #Warning.OP_WORK_MissingCnd := FALSE;
   END_IF;
END_REGION

REGION Network 14: <+>
END_REGION

REGION Network 15: << GESTIONE FERMI >>
END_REGION

REGION Network 16: P[1...6] DataIn
   RUNG wire#powerrail
      I_Contact( #HMI.Selection[1] )
      R_Coil( #Fermi[1].DataIn.PB.Rest )
      R_Coil( #Fermi[1].DataIn.PB.Work )
   END_RUNG
   RUNG wire#powerrail
      I_Contact( #HMI.Selection[2] )
      R_Coil( #Fermi[2].DataIn.PB.Rest )
      R_Coil( #Fermi[2].DataIn.PB.Work )
   END_RUNG
   RUNG wire#powerrail
      I_Contact( #HMI.Selection[3] )
      R_Coil( #Fermi[3].DataIn.PB.Rest )
      R_Coil( #Fermi[3].DataIn.PB.Work )
   END_RUNG
   RUNG wire#powerrail
      I_Contact( #HMI.Selection[4] )
      R_Coil( #Fermi[4].DataIn.PB.Rest )
      R_Coil( #Fermi[4].DataIn.PB.Work )
   END_RUNG
   RUNG wire#powerrail
      I_Contact( #HMI.Selection[5] )
      R_Coil( #Fermi[5].DataIn.PB.Rest )
      R_Coil( #Fermi[5].DataIn.PB.Work )
   END_RUNG
   RUNG wire#powerrail
      I_Contact( #HMI.Selection[6] )
      R_Coil( #Fermi[6].DataIn.PB.Rest )
      R_Coil( #Fermi[6].DataIn.PB.Work )
   END_RUNG
   // the same network as SCL:
   IF NOT #HMI.Selection[1] THEN
       #Fermi[1].DataIn.PB.Rest := FALSE;
       #Fermi[1].DataIn.PB.Work := FALSE;
   END_IF;
   IF NOT #HMI.Selection[2] THEN
       #Fermi[2].DataIn.PB.Rest := FALSE;
       #Fermi[2].DataIn.PB.Work := FALSE;
   END_IF;
   IF NOT #HMI.Selection[3] THEN
       #Fermi[3].DataIn.PB.Rest := FALSE;
       #Fermi[3].DataIn.PB.Work := FALSE;
   END_IF;
   IF NOT #HMI.Selection[4] THEN
       #Fermi[4].DataIn.PB.Rest := FALSE;
       #Fermi[4].DataIn.PB.Work := FALSE;
   END_IF;
   IF NOT #HMI.Selection[5] THEN
       #Fermi[5].DataIn.PB.Rest := FALSE;
       #Fermi[5].DataIn.PB.Work := FALSE;
   END_IF;
   IF NOT #HMI.Selection[6] THEN
       #Fermi[6].DataIn.PB.Rest := FALSE;
       #Fermi[6].DataIn.PB.Work := FALSE;
   END_IF;
END_REGION

REGION Network 17: P[1...6] CIn External alarm
   RUNG wire#powerrail
      Contact( FALSE )
      Coil( #Fermi[1].Cin.ExternalAlarms )
      Coil( #Fermi[2].Cin.ExternalAlarms )
      Coil( #Fermi[3].Cin.ExternalAlarms )
      Coil( #Fermi[4].Cin.ExternalAlarms )
      Coil( #Fermi[5].Cin.ExternalAlarms )
      Coil( #Fermi[6].Cin.ExternalAlarms )
   END_RUNG
   // the same network as SCL:
   #Fermi[1].Cin.ExternalAlarms := FALSE;
   #Fermi[2].Cin.ExternalAlarms := FALSE;
   #Fermi[3].Cin.ExternalAlarms := FALSE;
   #Fermi[4].Cin.ExternalAlarms := FALSE;
   #Fermi[5].Cin.ExternalAlarms := FALSE;
   #Fermi[6].Cin.ExternalAlarms := FALSE;
END_REGION

REGION Network 18: P[1...6] Cin REST Ext Enable
   RUNG wire#powerrail
      Contact( TRUE )
      wire#w1
      Coil( #Fermi[1].Cin.Rest_ExtEnable )
      Coil( #Fermi[2].Cin.Rest_ExtEnable )
      Coil( #Fermi[3].Cin.Rest_ExtEnable )
      Coil( #Fermi[4].Cin.Rest_ExtEnable )
      Coil( #Fermi[5].Cin.Rest_ExtEnable )
      Coil( #Fermi[6].Cin.Rest_ExtEnable )
   END_RUNG
   RUNG wire#powerrail
      Contact( #AreaInterface.Man )
      I_Contact( #CIn.Manager_Fermi.Control_ON )
      Contact( #Sts.OP_CanMoveFreely )
   END_RUNG wire#w1
   // the same network as SCL:
   #Fermi[1].Cin.Rest_ExtEnable := TRUE OR (#AreaInterface.Man AND NOT #CIn.Manager_Fermi.Control_ON AND #Sts.OP_CanMoveFreely);
   #Fermi[2].Cin.Rest_ExtEnable := TRUE OR (#AreaInterface.Man AND NOT #CIn.Manager_Fermi.Control_ON AND #Sts.OP_CanMoveFreely);
   #Fermi[3].Cin.Rest_ExtEnable := TRUE OR (#AreaInterface.Man AND NOT #CIn.Manager_Fermi.Control_ON AND #Sts.OP_CanMoveFreely);
   #Fermi[4].Cin.Rest_ExtEnable := TRUE OR (#AreaInterface.Man AND NOT #CIn.Manager_Fermi.Control_ON AND #Sts.OP_CanMoveFreely);
   #Fermi[5].Cin.Rest_ExtEnable := TRUE OR (#AreaInterface.Man AND NOT #CIn.Manager_Fermi.Control_ON AND #Sts.OP_CanMoveFreely);
   #Fermi[6].Cin.Rest_ExtEnable := TRUE OR (#AreaInterface.Man AND NOT #CIn.Manager_Fermi.Control_ON AND #Sts.OP_CanMoveFreely);
END_REGION

REGION Network 19: P[1...6] Cin WORK Ext Enable
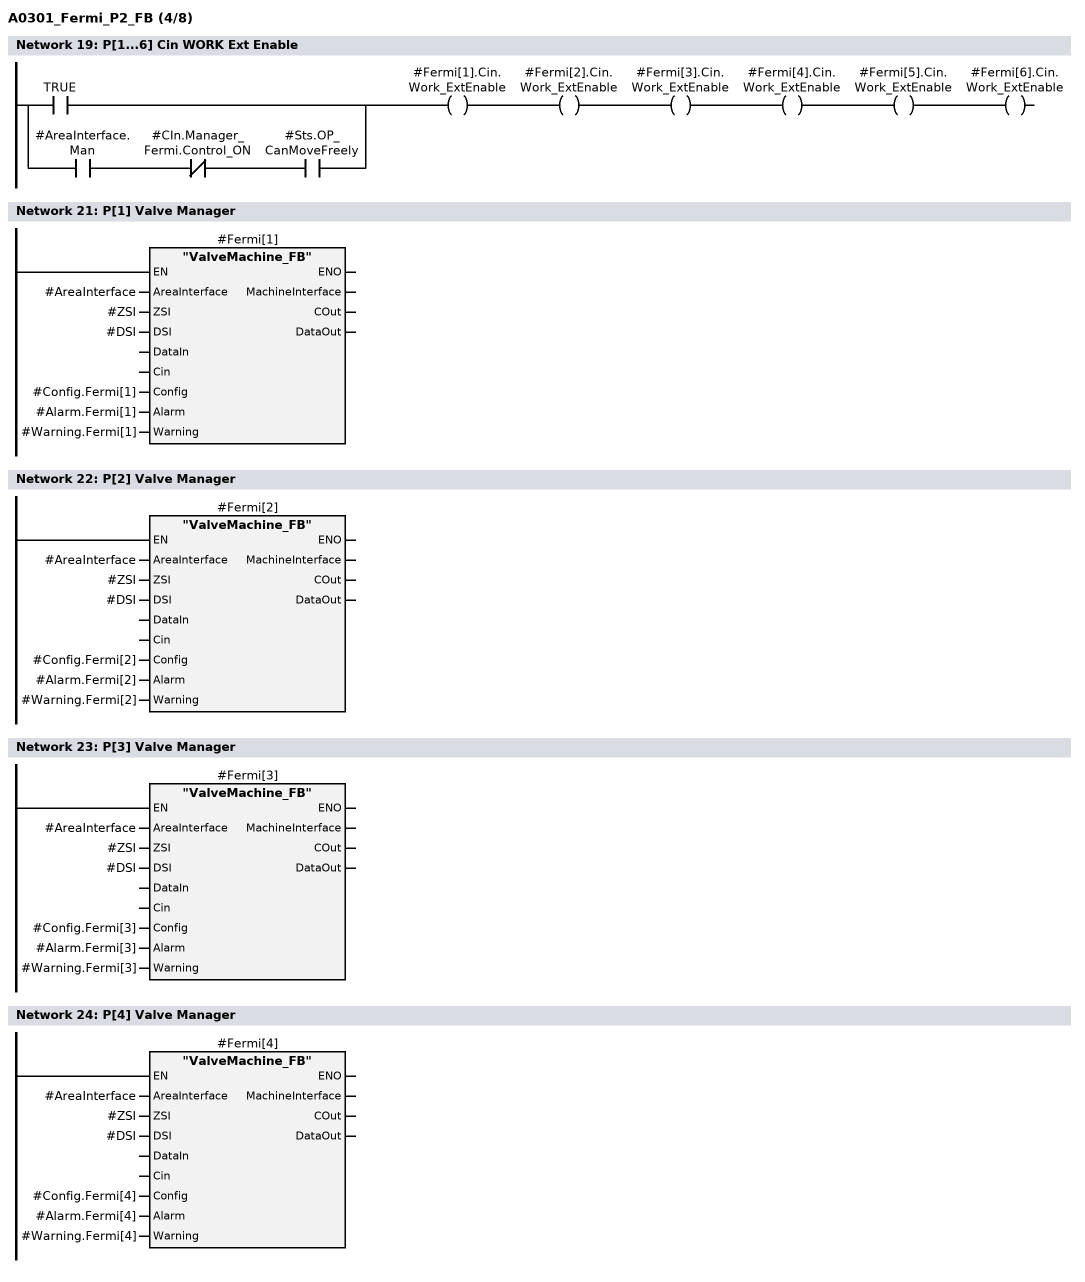
   RUNG wire#powerrail
      Contact( TRUE )
      wire#w1
      Coil( #Fermi[1].Cin.Work_ExtEnable )
      Coil( #Fermi[2].Cin.Work_ExtEnable )
      Coil( #Fermi[3].Cin.Work_ExtEnable )
      Coil( #Fermi[4].Cin.Work_ExtEnable )
      Coil( #Fermi[5].Cin.Work_ExtEnable )
      Coil( #Fermi[6].Cin.Work_ExtEnable )
   END_RUNG
   RUNG wire#powerrail
      Contact( #AreaInterface.Man )
      I_Contact( #CIn.Manager_Fermi.Control_ON )
      Contact( #Sts.OP_CanMoveFreely )
   END_RUNG wire#w1
   // the same network as SCL:
   #Fermi[1].Cin.Work_ExtEnable := TRUE OR (#AreaInterface.Man AND NOT #CIn.Manager_Fermi.Control_ON AND #Sts.OP_CanMoveFreely);
   #Fermi[2].Cin.Work_ExtEnable := TRUE OR (#AreaInterface.Man AND NOT #CIn.Manager_Fermi.Control_ON AND #Sts.OP_CanMoveFreely);
   #Fermi[3].Cin.Work_ExtEnable := TRUE OR (#AreaInterface.Man AND NOT #CIn.Manager_Fermi.Control_ON AND #Sts.OP_CanMoveFreely);
   #Fermi[4].Cin.Work_ExtEnable := TRUE OR (#AreaInterface.Man AND NOT #CIn.Manager_Fermi.Control_ON AND #Sts.OP_CanMoveFreely);
   #Fermi[5].Cin.Work_ExtEnable := TRUE OR (#AreaInterface.Man AND NOT #CIn.Manager_Fermi.Control_ON AND #Sts.OP_CanMoveFreely);
   #Fermi[6].Cin.Work_ExtEnable := TRUE OR (#AreaInterface.Man AND NOT #CIn.Manager_Fermi.Control_ON AND #Sts.OP_CanMoveFreely);
END_REGION

REGION Network 20: <+>
END_REGION

REGION Network 21: P[1] Valve Manager
   RUNG wire#powerrail
      #Fermi[1](AreaInterface := #AreaInterface, ZSI := #ZSI, DSI := #DSI, DataIn :=, Cin :=, Config := #Config.Fermi[1], Alarm := #Alarm.Fermi[1], Warning := #Warning.Fermi[1], MachineInterface =>, COut =>, DataOut =>)
   END_RUNG
   // the same network as SCL:
   #Fermi[1](AreaInterface := #AreaInterface,   // "ValveMachine_FB"
             ZSI := #ZSI,
             DSI := #DSI,
             Config := #Config.Fermi[1],
             Alarm := #Alarm.Fermi[1],
             Warning := #Warning.Fermi[1]);
END_REGION

REGION Network 22: P[2] Valve Manager
   RUNG wire#powerrail
      #Fermi[2](AreaInterface := #AreaInterface, ZSI := #ZSI, DSI := #DSI, DataIn :=, Cin :=, Config := #Config.Fermi[2], Alarm := #Alarm.Fermi[2], Warning := #Warning.Fermi[2], MachineInterface =>, COut =>, DataOut =>)
   END_RUNG
   // the same network as SCL:
   #Fermi[2](AreaInterface := #AreaInterface,   // "ValveMachine_FB"
             ZSI := #ZSI,
             DSI := #DSI,
             Config := #Config.Fermi[2],
             Alarm := #Alarm.Fermi[2],
             Warning := #Warning.Fermi[2]);
END_REGION

REGION Network 23: P[3] Valve Manager
   RUNG wire#powerrail
      #Fermi[3](AreaInterface := #AreaInterface, ZSI := #ZSI, DSI := #DSI, DataIn :=, Cin :=, Config := #Config.Fermi[3], Alarm := #Alarm.Fermi[3], Warning := #Warning.Fermi[3], MachineInterface =>, COut =>, DataOut =>)
   END_RUNG
   // the same network as SCL:
   #Fermi[3](AreaInterface := #AreaInterface,   // "ValveMachine_FB"
             ZSI := #ZSI,
             DSI := #DSI,
             Config := #Config.Fermi[3],
             Alarm := #Alarm.Fermi[3],
             Warning := #Warning.Fermi[3]);
END_REGION

REGION Network 24: P[4] Valve Manager
   RUNG wire#powerrail
      #Fermi[4](AreaInterface := #AreaInterface, ZSI := #ZSI, DSI := #DSI, DataIn :=, Cin :=, Config := #Config.Fermi[4], Alarm := #Alarm.Fermi[4], Warning := #Warning.Fermi[4], MachineInterface =>, COut =>, DataOut =>)
   END_RUNG
   // the same network as SCL:
   #Fermi[4](AreaInterface := #AreaInterface,   // "ValveMachine_FB"
             ZSI := #ZSI,
             DSI := #DSI,
             Config := #Config.Fermi[4],
             Alarm := #Alarm.Fermi[4],
             Warning := #Warning.Fermi[4]);
END_REGION

REGION Network 25: P[5] Valve Manager
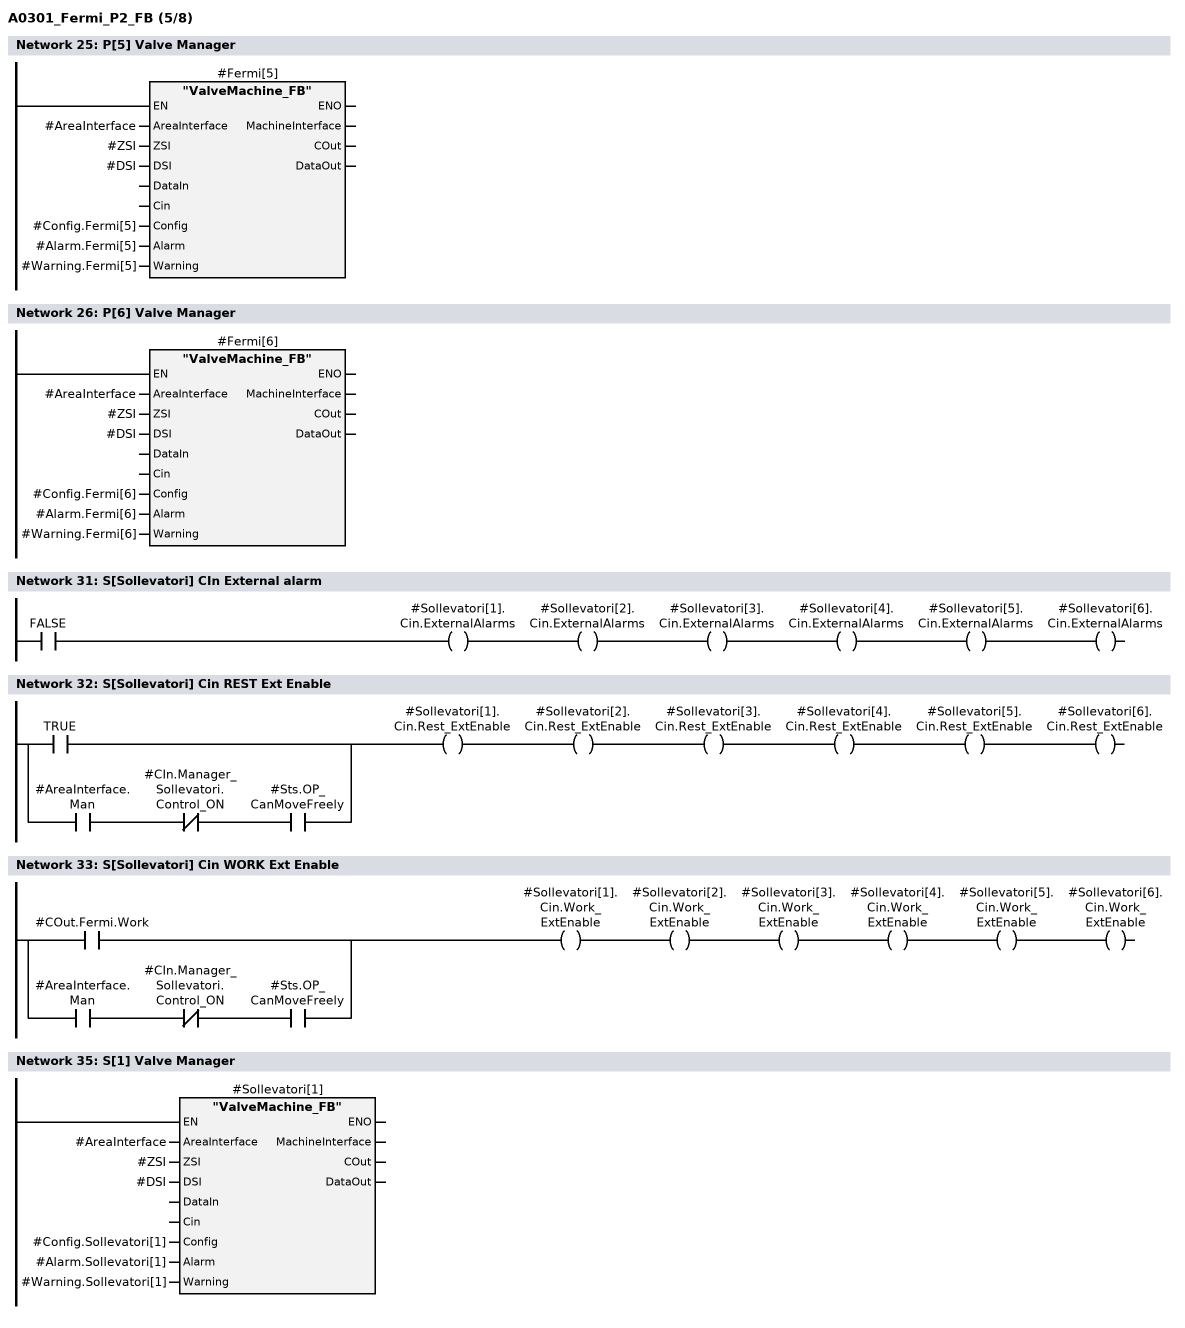
   RUNG wire#powerrail
      #Fermi[5](AreaInterface := #AreaInterface, ZSI := #ZSI, DSI := #DSI, DataIn :=, Cin :=, Config := #Config.Fermi[5], Alarm := #Alarm.Fermi[5], Warning := #Warning.Fermi[5], MachineInterface =>, COut =>, DataOut =>)
   END_RUNG
   // the same network as SCL:
   #Fermi[5](AreaInterface := #AreaInterface,   // "ValveMachine_FB"
             ZSI := #ZSI,
             DSI := #DSI,
             Config := #Config.Fermi[5],
             Alarm := #Alarm.Fermi[5],
             Warning := #Warning.Fermi[5]);
END_REGION

REGION Network 26: P[6] Valve Manager
   RUNG wire#powerrail
      #Fermi[6](AreaInterface := #AreaInterface, ZSI := #ZSI, DSI := #DSI, DataIn :=, Cin :=, Config := #Config.Fermi[6], Alarm := #Alarm.Fermi[6], Warning := #Warning.Fermi[6], MachineInterface =>, COut =>, DataOut =>)
   END_RUNG
   // the same network as SCL:
   #Fermi[6](AreaInterface := #AreaInterface,   // "ValveMachine_FB"
             ZSI := #ZSI,
             DSI := #DSI,
             Config := #Config.Fermi[6],
             Alarm := #Alarm.Fermi[6],
             Warning := #Warning.Fermi[6]);
END_REGION

REGION Network 27: <+>
END_REGION

REGION Network 28 (SCL): P[1...6] COut Fermi
   REGION COut STANDSTILL Fermi
       // Controllo uscita COut STANDSTILL in base allo stato di tutti i Pin
       IF  #Fermi[1].Sts.Standstill AND
           #Fermi[2].Sts.Standstill AND
           #Fermi[3].Sts.Standstill AND
           #Fermi[4].Sts.Standstill AND
           #Fermi[5].Sts.Standstill AND
           #Fermi[6].Sts.Standstill THEN
           #COut.Fermi.Standstill := TRUE;
       ELSE
           #COut.Fermi.Standstill := FALSE;
       END_IF;
   END_REGION ;


   REGION COut AT REST #Fermi
       // Controllo uscita COut AT_REST in base allo stato di tutti i Pin
       IF  #Fermi[1].COut.Rest OR #Fermi[1].DataIn.Rest_Ls[1] AND
           #Fermi[2].COut.Rest OR #Fermi[2].DataIn.Rest_Ls[1] AND
           #Fermi[3].COut.Rest OR #Fermi[3].DataIn.Rest_Ls[1] AND
           #Fermi[4].COut.Rest OR #Fermi[4].DataIn.Rest_Ls[1] AND
           #Fermi[5].COut.Rest OR #Fermi[5].DataIn.Rest_Ls[1] AND
           #Fermi[6].COut.Rest OR #Fermi[6].DataIn.Rest_Ls[1] THEN
           #COut.Fermi.Rest := 1;
       ELSE
           #COut.Fermi.Rest := 0;
       END_IF;
   END_REGION ;

   REGION COut AT WORK Fermi
       // Controllo uscita COut AT_WORK in base allo stato di tutti i Pin
       IF  #Fermi[1].COut.Work AND
           #Fermi[2].COut.Work AND
           #Fermi[3].COut.Work AND
           #Fermi[4].COut.Work AND
           #Fermi[5].COut.Work AND
           #Fermi[6].COut.Work THEN
           #COut.Fermi.Work := 1;
       ELSE
           #COut.Fermi.Work := 0;
       END_IF;
   END_REGION ;
END_REGION

REGION Network 30: <<<< GESTIONE SOLLEVATORE - SemiGuscio >>>
END_REGION

REGION Network 31: S[Sollevatori] CIn External alarm
   RUNG wire#powerrail
      Contact( FALSE )
      Coil( #Sollevatori[1].Cin.ExternalAlarms )
      Coil( #Sollevatori[2].Cin.ExternalAlarms )
      Coil( #Sollevatori[3].Cin.ExternalAlarms )
      Coil( #Sollevatori[4].Cin.ExternalAlarms )
      Coil( #Sollevatori[5].Cin.ExternalAlarms )
      Coil( #Sollevatori[6].Cin.ExternalAlarms )
   END_RUNG
   // the same network as SCL:
   #Sollevatori[1].Cin.ExternalAlarms := FALSE;
   #Sollevatori[2].Cin.ExternalAlarms := FALSE;
   #Sollevatori[3].Cin.ExternalAlarms := FALSE;
   #Sollevatori[4].Cin.ExternalAlarms := FALSE;
   #Sollevatori[5].Cin.ExternalAlarms := FALSE;
   #Sollevatori[6].Cin.ExternalAlarms := FALSE;
END_REGION

REGION Network 32: S[Sollevatori] Cin REST Ext Enable
   RUNG wire#powerrail
      Contact( TRUE )
      wire#w1
      Coil( #Sollevatori[1].Cin.Rest_ExtEnable )
      Coil( #Sollevatori[2].Cin.Rest_ExtEnable )
      Coil( #Sollevatori[3].Cin.Rest_ExtEnable )
      Coil( #Sollevatori[4].Cin.Rest_ExtEnable )
      Coil( #Sollevatori[5].Cin.Rest_ExtEnable )
      Coil( #Sollevatori[6].Cin.Rest_ExtEnable )
   END_RUNG
   RUNG wire#powerrail
      Contact( #AreaInterface.Man )
      I_Contact( #CIn.Manager_Sollevatori.Control_ON )
      Contact( #Sts.OP_CanMoveFreely )
   END_RUNG wire#w1
   // the same network as SCL:
   #Sollevatori[1].Cin.Rest_ExtEnable := TRUE OR (#AreaInterface.Man AND NOT #CIn.Manager_Sollevatori.Control_ON AND #Sts.OP_CanMoveFreely);
   #Sollevatori[2].Cin.Rest_ExtEnable := TRUE OR (#AreaInterface.Man AND NOT #CIn.Manager_Sollevatori.Control_ON AND #Sts.OP_CanMoveFreely);
   #Sollevatori[3].Cin.Rest_ExtEnable := TRUE OR (#AreaInterface.Man AND NOT #CIn.Manager_Sollevatori.Control_ON AND #Sts.OP_CanMoveFreely);
   #Sollevatori[4].Cin.Rest_ExtEnable := TRUE OR (#AreaInterface.Man AND NOT #CIn.Manager_Sollevatori.Control_ON AND #Sts.OP_CanMoveFreely);
   #Sollevatori[5].Cin.Rest_ExtEnable := TRUE OR (#AreaInterface.Man AND NOT #CIn.Manager_Sollevatori.Control_ON AND #Sts.OP_CanMoveFreely);
   #Sollevatori[6].Cin.Rest_ExtEnable := TRUE OR (#AreaInterface.Man AND NOT #CIn.Manager_Sollevatori.Control_ON AND #Sts.OP_CanMoveFreely);
END_REGION

REGION Network 33: S[Sollevatori] Cin WORK Ext Enable
   RUNG wire#powerrail
      Contact( #COut.Fermi.Work )
      wire#w1
      Coil( #Sollevatori[1].Cin.Work_ExtEnable )
      Coil( #Sollevatori[2].Cin.Work_ExtEnable )
      Coil( #Sollevatori[3].Cin.Work_ExtEnable )
      Coil( #Sollevatori[4].Cin.Work_ExtEnable )
      Coil( #Sollevatori[5].Cin.Work_ExtEnable )
      Coil( #Sollevatori[6].Cin.Work_ExtEnable )
   END_RUNG
   RUNG wire#powerrail
      Contact( #AreaInterface.Man )
      I_Contact( #CIn.Manager_Sollevatori.Control_ON )
      Contact( #Sts.OP_CanMoveFreely )
   END_RUNG wire#w1
   // the same network as SCL:
   #Sollevatori[1].Cin.Work_ExtEnable := #COut.Fermi.Work OR (#AreaInterface.Man AND NOT #CIn.Manager_Sollevatori.Control_ON AND #Sts.OP_CanMoveFreely);
   #Sollevatori[2].Cin.Work_ExtEnable := #COut.Fermi.Work OR (#AreaInterface.Man AND NOT #CIn.Manager_Sollevatori.Control_ON AND #Sts.OP_CanMoveFreely);
   #Sollevatori[3].Cin.Work_ExtEnable := #COut.Fermi.Work OR (#AreaInterface.Man AND NOT #CIn.Manager_Sollevatori.Control_ON AND #Sts.OP_CanMoveFreely);
   #Sollevatori[4].Cin.Work_ExtEnable := #COut.Fermi.Work OR (#AreaInterface.Man AND NOT #CIn.Manager_Sollevatori.Control_ON AND #Sts.OP_CanMoveFreely);
   #Sollevatori[5].Cin.Work_ExtEnable := #COut.Fermi.Work OR (#AreaInterface.Man AND NOT #CIn.Manager_Sollevatori.Control_ON AND #Sts.OP_CanMoveFreely);
   #Sollevatori[6].Cin.Work_ExtEnable := #COut.Fermi.Work OR (#AreaInterface.Man AND NOT #CIn.Manager_Sollevatori.Control_ON AND #Sts.OP_CanMoveFreely);
END_REGION

REGION Network 34: <+>
END_REGION

REGION Network 35: S[1] Valve Manager
   RUNG wire#powerrail
      #Sollevatori[1](AreaInterface := #AreaInterface, ZSI := #ZSI, DSI := #DSI, DataIn :=, Cin :=, Config := #Config.Sollevatori[1], Alarm := #Alarm.Sollevatori[1], Warning := #Warning.Sollevatori[1], MachineInterface =>, COut =>, DataOut =>)
   END_RUNG
   // the same network as SCL:
   #Sollevatori[1](AreaInterface := #AreaInterface,   // "ValveMachine_FB"
                   ZSI := #ZSI,
                   DSI := #DSI,
                   Config := #Config.Sollevatori[1],
                   Alarm := #Alarm.Sollevatori[1],
                   Warning := #Warning.Sollevatori[1]);
END_REGION

REGION Network 36: S[2] Valve Manager
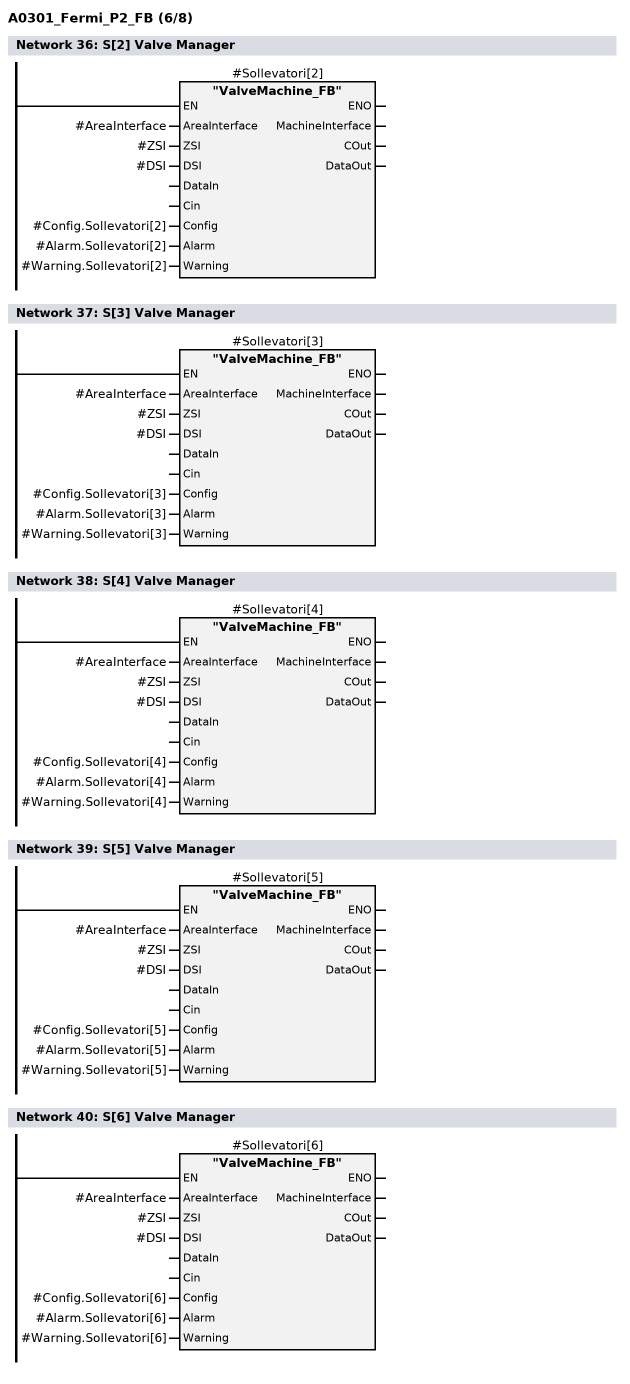
   RUNG wire#powerrail
      #Sollevatori[2](AreaInterface := #AreaInterface, ZSI := #ZSI, DSI := #DSI, DataIn :=, Cin :=, Config := #Config.Sollevatori[2], Alarm := #Alarm.Sollevatori[2], Warning := #Warning.Sollevatori[2], MachineInterface =>, COut =>, DataOut =>)
   END_RUNG
   // the same network as SCL:
   #Sollevatori[2](AreaInterface := #AreaInterface,   // "ValveMachine_FB"
                   ZSI := #ZSI,
                   DSI := #DSI,
                   Config := #Config.Sollevatori[2],
                   Alarm := #Alarm.Sollevatori[2],
                   Warning := #Warning.Sollevatori[2]);
END_REGION

REGION Network 37: S[3] Valve Manager
   RUNG wire#powerrail
      #Sollevatori[3](AreaInterface := #AreaInterface, ZSI := #ZSI, DSI := #DSI, DataIn :=, Cin :=, Config := #Config.Sollevatori[3], Alarm := #Alarm.Sollevatori[3], Warning := #Warning.Sollevatori[3], MachineInterface =>, COut =>, DataOut =>)
   END_RUNG
   // the same network as SCL:
   #Sollevatori[3](AreaInterface := #AreaInterface,   // "ValveMachine_FB"
                   ZSI := #ZSI,
                   DSI := #DSI,
                   Config := #Config.Sollevatori[3],
                   Alarm := #Alarm.Sollevatori[3],
                   Warning := #Warning.Sollevatori[3]);
END_REGION

REGION Network 38: S[4] Valve Manager
   RUNG wire#powerrail
      #Sollevatori[4](AreaInterface := #AreaInterface, ZSI := #ZSI, DSI := #DSI, DataIn :=, Cin :=, Config := #Config.Sollevatori[4], Alarm := #Alarm.Sollevatori[4], Warning := #Warning.Sollevatori[4], MachineInterface =>, COut =>, DataOut =>)
   END_RUNG
   // the same network as SCL:
   #Sollevatori[4](AreaInterface := #AreaInterface,   // "ValveMachine_FB"
                   ZSI := #ZSI,
                   DSI := #DSI,
                   Config := #Config.Sollevatori[4],
                   Alarm := #Alarm.Sollevatori[4],
                   Warning := #Warning.Sollevatori[4]);
END_REGION

REGION Network 39: S[5] Valve Manager
   RUNG wire#powerrail
      #Sollevatori[5](AreaInterface := #AreaInterface, ZSI := #ZSI, DSI := #DSI, DataIn :=, Cin :=, Config := #Config.Sollevatori[5], Alarm := #Alarm.Sollevatori[5], Warning := #Warning.Sollevatori[5], MachineInterface =>, COut =>, DataOut =>)
   END_RUNG
   // the same network as SCL:
   #Sollevatori[5](AreaInterface := #AreaInterface,   // "ValveMachine_FB"
                   ZSI := #ZSI,
                   DSI := #DSI,
                   Config := #Config.Sollevatori[5],
                   Alarm := #Alarm.Sollevatori[5],
                   Warning := #Warning.Sollevatori[5]);
END_REGION

REGION Network 40: S[6] Valve Manager
   RUNG wire#powerrail
      #Sollevatori[6](AreaInterface := #AreaInterface, ZSI := #ZSI, DSI := #DSI, DataIn :=, Cin :=, Config := #Config.Sollevatori[6], Alarm := #Alarm.Sollevatori[6], Warning := #Warning.Sollevatori[6], MachineInterface =>, COut =>, DataOut =>)
   END_RUNG
   // the same network as SCL:
   #Sollevatori[6](AreaInterface := #AreaInterface,   // "ValveMachine_FB"
                   ZSI := #ZSI,
                   DSI := #DSI,
                   Config := #Config.Sollevatori[6],
                   Alarm := #Alarm.Sollevatori[6],
                   Warning := #Warning.Sollevatori[6]);
END_REGION

REGION Network 41: <+>
END_REGION

REGION Network 42 (SCL): S[Sollevatori] COut
   REGION COut STANDSTILL Sollevatori
       // Controllo uscita COut STANDSTILL in base allo stato di tutti i pistoni
       IF  #Sollevatori[1].Sts.Standstill AND
           #Sollevatori[2].Sts.Standstill AND
           #Sollevatori[3].Sts.Standstill AND
           #Sollevatori[4].Sts.Standstill AND
           #Sollevatori[5].Sts.Standstill AND
           #Sollevatori[6].Sts.Standstill THEN
           #COut.Sollevatori.Standstill := TRUE;
       ELSE
           #COut.Sollevatori.Standstill := FALSE;
       END_IF;
   END_REGION ;


   REGION COut AT REST Sollevatori
       // Controllo uscita COut AT_REST in base allo stato di tutti i pistoni
       IF  #Sollevatori[1].COut.Rest OR #Sollevatori[1].DataIn.Rest_Ls[1] AND
           #Sollevatori[2].COut.Rest OR #Sollevatori[2].DataIn.Rest_Ls[1] AND
           #Sollevatori[3].COut.Rest OR #Sollevatori[3].DataIn.Rest_Ls[1] AND
           #Sollevatori[4].COut.Rest OR #Sollevatori[4].DataIn.Rest_Ls[1] AND
           #Sollevatori[5].COut.Rest OR #Sollevatori[5].DataIn.Rest_Ls[1] AND
           #Sollevatori[6].COut.Rest OR #Sollevatori[6].DataIn.Rest_Ls[1] THEN
           #COut.Sollevatori.Rest := 1;
       ELSE
           #COut.Sollevatori.Rest := 0;
       END_IF;
   END_REGION ;

   REGION COut AT WORK Sollevatori
       // Controllo uscita COut AT_WORK in base allo stato di tutti i pistoni
       IF  #Sollevatori[1].COut.Work AND
           #Sollevatori[2].COut.Work AND
           #Sollevatori[3].COut.Work AND
           #Sollevatori[4].COut.Work AND
           #Sollevatori[5].COut.Work AND
           #Sollevatori[6].COut.Work THEN
           #COut.Sollevatori.Work := 1;
       ELSE
           #COut.Sollevatori.Work := 0;
       END_IF;
   END_REGION ;
END_REGION

REGION Network 44: Fermi + Sollevatori - Accumulativo status Alarm
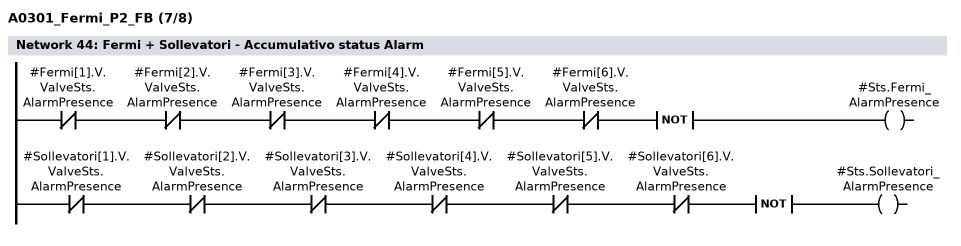
   RUNG wire#powerrail
      I_Contact( #Fermi[1].V.ValveSts.AlarmPresence )
      I_Contact( #Fermi[2].V.ValveSts.AlarmPresence )
      I_Contact( #Fermi[3].V.ValveSts.AlarmPresence )
      I_Contact( #Fermi[4].V.ValveSts.AlarmPresence )
      I_Contact( #Fermi[5].V.ValveSts.AlarmPresence )
      I_Contact( #Fermi[6].V.ValveSts.AlarmPresence )
      Not()
      Coil( #Sts.Fermi_AlarmPresence )
   END_RUNG
   RUNG wire#powerrail
      I_Contact( #Sollevatori[1].V.ValveSts.AlarmPresence )
      I_Contact( #Sollevatori[2].V.ValveSts.AlarmPresence )
      I_Contact( #Sollevatori[3].V.ValveSts.AlarmPresence )
      I_Contact( #Sollevatori[4].V.ValveSts.AlarmPresence )
      I_Contact( #Sollevatori[5].V.ValveSts.AlarmPresence )
      I_Contact( #Sollevatori[6].V.ValveSts.AlarmPresence )
      Not()
      Coil( #Sts.Sollevatori_AlarmPresence )
   END_RUNG
   // the same network as SCL:
   #Sts.Fermi_AlarmPresence := NOT (NOT #Fermi[1].V.ValveSts.AlarmPresence AND NOT #Fermi[2].V.ValveSts.AlarmPresence AND NOT #Fermi[3].V.ValveSts.AlarmPresence AND NOT #Fermi[4].V.ValveSts.AlarmPresence AND NOT #Fermi[5].V.ValveSts.AlarmPresence AND NOT #Fermi[6].V.ValveSts.AlarmPresence);
   #Sts.Sollevatori_AlarmPresence := NOT (NOT #Sollevatori[1].V.ValveSts.AlarmPresence AND NOT #Sollevatori[2].V.ValveSts.AlarmPresence AND NOT #Sollevatori[3].V.ValveSts.AlarmPresence AND NOT #Sollevatori[4].V.ValveSts.AlarmPresence AND NOT #Sollevatori[5].V.ValveSts.AlarmPresence AND NOT #Sollevatori[6].V.ValveSts.AlarmPresence);
END_REGION

REGION Network 45 (SCL): HMI STATUS - Postazione
   // Area dati appoggio per HMI
   // FERMI POS.2
   #HMI.FermiSts.Standstill := #COut.Fermi.Standstill;
   #HMI.FermiSts.Rest := #COut.Fermi.Rest;
   #HMI.FermiSts.Work := #COut.Fermi.Work;
   #HMI.FermiSts.AlarmPresence := #Sts.Fermi_AlarmPresence;

   // SOLLEVATORI POS.2
   #HMI.SollevatoriSts.Standstill := #COut.Sollevatori.Standstill;
   #HMI.SollevatoriSts.Rest := #COut.Sollevatori.Rest;
   #HMI.SollevatoriSts.Work := #COut.Sollevatori.Work;
   #HMI.SollevatoriSts.AlarmPresence := #Sts.Sollevatori_AlarmPresence;
END_REGION

REGION Network 47: << MAIN MACHINE STATUS >>
END_REGION

REGION Network 48: Machine interface
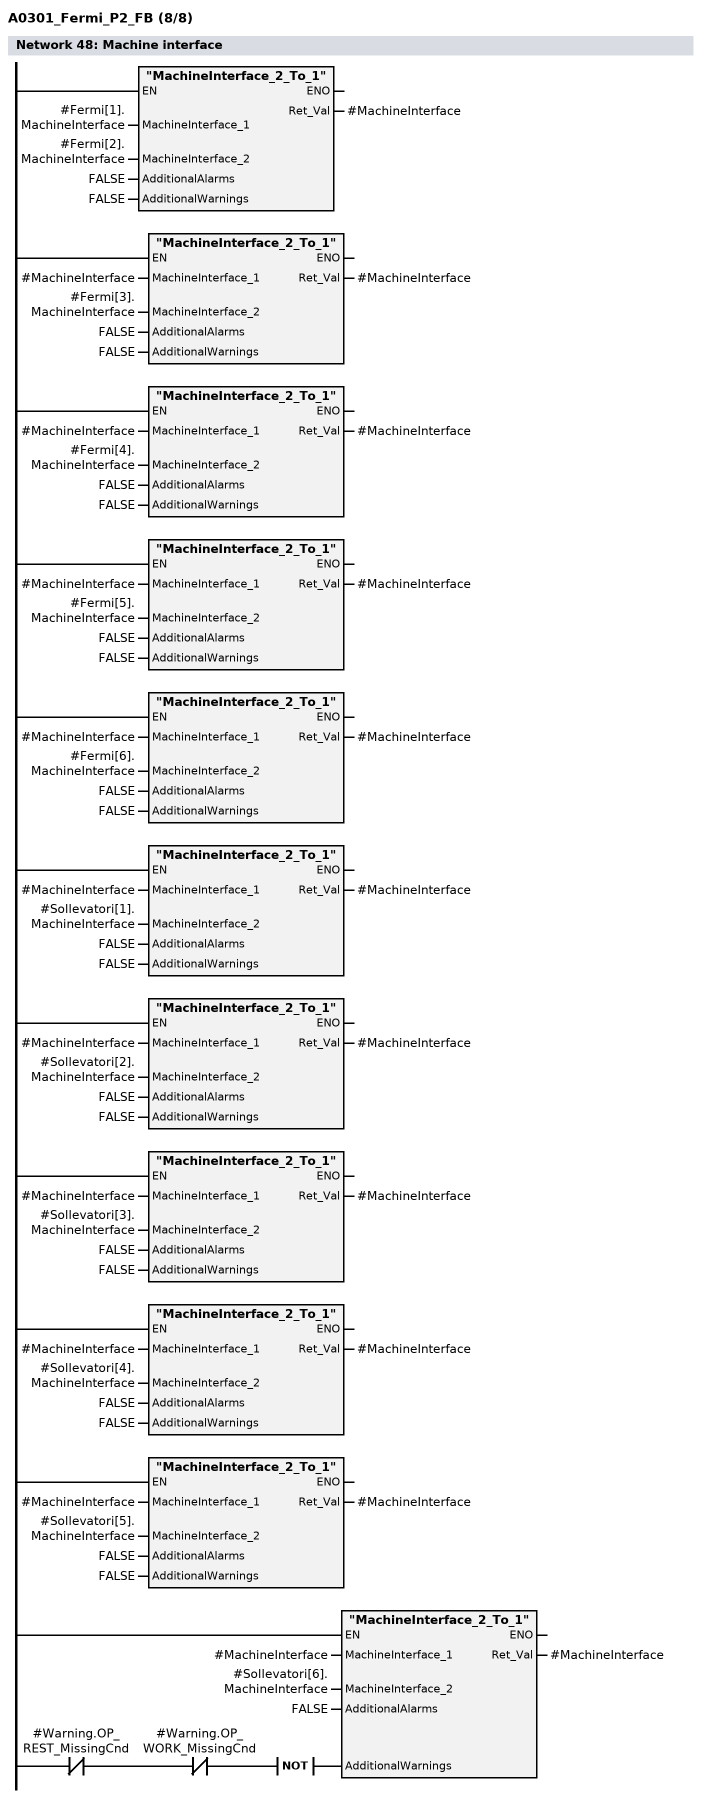
   RUNG wire#powerrail
      "MachineInterface_2_To_1"(MachineInterface_1 := #Fermi[1].MachineInterface, MachineInterface_2 := #Fermi[2].MachineInterface, AdditionalAlarms := FALSE, AdditionalWarnings := FALSE, Ret_Val => #MachineInterface)
   END_RUNG
   RUNG wire#powerrail
      "MachineInterface_2_To_1"(MachineInterface_1 := #MachineInterface, MachineInterface_2 := #Fermi[3].MachineInterface, AdditionalAlarms := FALSE, AdditionalWarnings := FALSE, Ret_Val => #MachineInterface)
   END_RUNG
   RUNG wire#powerrail
      "MachineInterface_2_To_1"(MachineInterface_1 := #MachineInterface, MachineInterface_2 := #Fermi[4].MachineInterface, AdditionalAlarms := FALSE, AdditionalWarnings := FALSE, Ret_Val => #MachineInterface)
   END_RUNG
   RUNG wire#powerrail
      "MachineInterface_2_To_1"(MachineInterface_1 := #MachineInterface, MachineInterface_2 := #Fermi[5].MachineInterface, AdditionalAlarms := FALSE, AdditionalWarnings := FALSE, Ret_Val => #MachineInterface)
   END_RUNG
   RUNG wire#powerrail
      "MachineInterface_2_To_1"(MachineInterface_1 := #MachineInterface, MachineInterface_2 := #Fermi[6].MachineInterface, AdditionalAlarms := FALSE, AdditionalWarnings := FALSE, Ret_Val => #MachineInterface)
   END_RUNG
   RUNG wire#powerrail
      "MachineInterface_2_To_1"(MachineInterface_1 := #MachineInterface, MachineInterface_2 := #Sollevatori[1].MachineInterface, AdditionalAlarms := FALSE, AdditionalWarnings := FALSE, Ret_Val => #MachineInterface)
   END_RUNG
   RUNG wire#powerrail
      "MachineInterface_2_To_1"(MachineInterface_1 := #MachineInterface, MachineInterface_2 := #Sollevatori[2].MachineInterface, AdditionalAlarms := FALSE, AdditionalWarnings := FALSE, Ret_Val => #MachineInterface)
   END_RUNG
   RUNG wire#powerrail
      "MachineInterface_2_To_1"(MachineInterface_1 := #MachineInterface, MachineInterface_2 := #Sollevatori[3].MachineInterface, AdditionalAlarms := FALSE, AdditionalWarnings := FALSE, Ret_Val => #MachineInterface)
   END_RUNG
   RUNG wire#powerrail
      "MachineInterface_2_To_1"(MachineInterface_1 := #MachineInterface, MachineInterface_2 := #Sollevatori[4].MachineInterface, AdditionalAlarms := FALSE, AdditionalWarnings := FALSE, Ret_Val => #MachineInterface)
   END_RUNG
   RUNG wire#powerrail
      "MachineInterface_2_To_1"(MachineInterface_1 := #MachineInterface, MachineInterface_2 := #Sollevatori[5].MachineInterface, AdditionalAlarms := FALSE, AdditionalWarnings := FALSE, Ret_Val => #MachineInterface)
   END_RUNG
   RUNG wire#powerrail
      "MachineInterface_2_To_1"(AdditionalWarnings := wire#w1, MachineInterface_1 := #MachineInterface, MachineInterface_2 := #Sollevatori[6].MachineInterface, AdditionalAlarms := FALSE, Ret_Val => #MachineInterface)
   END_RUNG
   RUNG wire#powerrail
      I_Contact( #Warning.OP_REST_MissingCnd )
      I_Contact( #Warning.OP_WORK_MissingCnd )
      Not()
   END_RUNG wire#w1
   // the same network as SCL:
   #MachineInterface := "MachineInterface_2_To_1"(MachineInterface_1 := #Fermi[1].MachineInterface,
                           MachineInterface_2 := #Fermi[2].MachineInterface,
                           AdditionalAlarms := FALSE,
                           AdditionalWarnings := FALSE);
   #MachineInterface := "MachineInterface_2_To_1"(MachineInterface_1 := #MachineInterface,
                           MachineInterface_2 := #Fermi[3].MachineInterface,
                           AdditionalAlarms := FALSE,
                           AdditionalWarnings := FALSE);
   #MachineInterface := "MachineInterface_2_To_1"(MachineInterface_1 := #MachineInterface,
                           MachineInterface_2 := #Fermi[4].MachineInterface,
                           AdditionalAlarms := FALSE,
                           AdditionalWarnings := FALSE);
   #MachineInterface := "MachineInterface_2_To_1"(MachineInterface_1 := #MachineInterface,
                           MachineInterface_2 := #Fermi[5].MachineInterface,
                           AdditionalAlarms := FALSE,
                           AdditionalWarnings := FALSE);
   #MachineInterface := "MachineInterface_2_To_1"(MachineInterface_1 := #MachineInterface,
                           MachineInterface_2 := #Fermi[6].MachineInterface,
                           AdditionalAlarms := FALSE,
                           AdditionalWarnings := FALSE);
   #MachineInterface := "MachineInterface_2_To_1"(MachineInterface_1 := #MachineInterface,
                           MachineInterface_2 := #Sollevatori[1].MachineInterface,
                           AdditionalAlarms := FALSE,
                           AdditionalWarnings := FALSE);
   #MachineInterface := "MachineInterface_2_To_1"(MachineInterface_1 := #MachineInterface,
                           MachineInterface_2 := #Sollevatori[2].MachineInterface,
                           AdditionalAlarms := FALSE,
                           AdditionalWarnings := FALSE);
   #MachineInterface := "MachineInterface_2_To_1"(MachineInterface_1 := #MachineInterface,
                           MachineInterface_2 := #Sollevatori[3].MachineInterface,
                           AdditionalAlarms := FALSE,
                           AdditionalWarnings := FALSE);
   #MachineInterface := "MachineInterface_2_To_1"(MachineInterface_1 := #MachineInterface,
                           MachineInterface_2 := #Sollevatori[4].MachineInterface,
                           AdditionalAlarms := FALSE,
                           AdditionalWarnings := FALSE);
   #MachineInterface := "MachineInterface_2_To_1"(MachineInterface_1 := #MachineInterface,
                           MachineInterface_2 := #Sollevatori[5].MachineInterface,
                           AdditionalAlarms := FALSE,
                           AdditionalWarnings := FALSE);
   #MachineInterface := "MachineInterface_2_To_1"(MachineInterface_1 := #MachineInterface,
                           MachineInterface_2 := #Sollevatori[6].MachineInterface,
                           AdditionalAlarms := FALSE,
                           AdditionalWarnings := NOT (NOT #Warning.OP_REST_MissingCnd AND NOT #Warning.OP_WORK_MissingCnd));
END_REGION
END_FUNCTION_BLOCK

FUNCTION "A0301_Fermi_P3_CALL" : Void   // FC120, LAD
// stored: SetENOAutomatically false
BEGIN

REGION Network 1 (SCL): << TRASFERIMENTO stati CIn del blocco >>
   // TRASFERIMENTO #CIn MANAGER
   "A0301_Fermi_P3".CIn.Manager := "A0301_Manager".COut.P3.Fermi;
   //
   "A0301_Fermi_P3".CIn.SemiAut := "A0301_Manager".DataIn.SemiAut_Pb;

   // Trasferimento status alla Stazione P2 da COut a Cin delle stazioni successive
   "A0301_Fermi_P3".CIn.P2.Fermi := "A0301_Fermi_P2".COut.Fermi;

   // Trasferimento status alla Stazione P3 da COut a Cin del sollevatore P2
   "A0301_Fermi_P3".CIn.P2.Sollevatore := "A0301_Fermi_P2".COut.Sollevatori;

   // Trasferimenti status lettura posizioni Trasporto al Cin delle stazioni
   "A0301_Fermi_P3".CIn.Trasporto := "A0301_Trasporto".COut.Ax;
END_REGION

REGION Network 2 (SCL): << TRASFERIMENTO stati DataIn >>
   // SOSTITUIRE SYS.BAYPASS
   // TRASFERIMENTO #DataIn STATI BUTTON STAZIONE P3

   REGION TRASFERIMENTO DataIn DIGITAL INPUT dei LIMIT SWITCH

       // Trasferimento ingressi digitali Limit Switch Fermi P3
       // 
       "A0301_Fermi_P3".Fermi[1].DataIn.Rest_Ls[1] := "A0301_CinghiaTrasporto_1.2_Ls_Rest_1";
       "A0301_Fermi_P3".Fermi[2].DataIn.Rest_Ls[1] := "A0301_CinghiaTrasporto_2.2_Ls_Rest_1";
       "A0301_Fermi_P3".Fermi[3].DataIn.Rest_Ls[1] := "A0301_CinghiaTrasporto_3.2_Ls_Rest_1";
       "A0301_Fermi_P3".Fermi[4].DataIn.Rest_Ls[1] := "A0301_CinghiaTrasporto_4.2_Ls_Rest_1";
       "A0301_Fermi_P3".Fermi[5].DataIn.Rest_Ls[1] := "A0301_CinghiaTrasporto_5.2_Ls_Rest_1";
       "A0301_Fermi_P3".Fermi[6].DataIn.Rest_Ls[1] := "A0301_CinghiaTrasporto_6.2_Ls_Rest_1";

   END_REGION ;
END_REGION

REGION Network 3: DataIn - Fermi
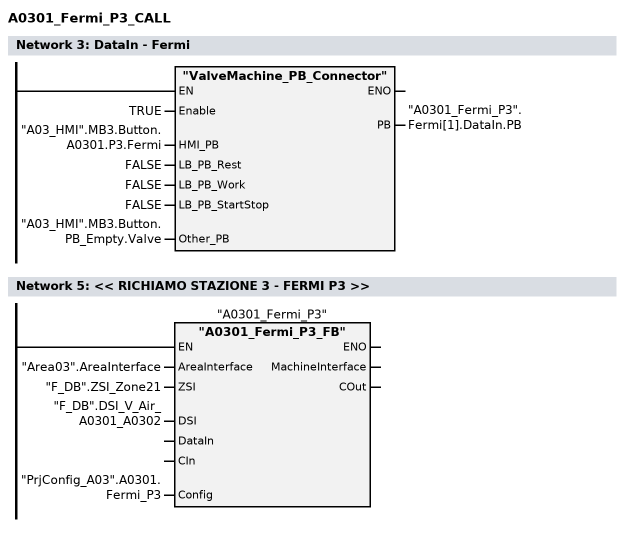
   RUNG wire#powerrail
      "ValveMachine_PB_Connector"(Enable := TRUE, HMI_PB := "A03_HMI".MB3.Button.A0301.P3.Fermi, LB_PB_Rest := FALSE, LB_PB_Work := FALSE, LB_PB_StartStop := FALSE, Other_PB := "A03_HMI".MB3.Button.PB_Empty.Valve, PB => "A0301_Fermi_P3".Fermi[1].DataIn.PB)
   END_RUNG
   // the same network as SCL:
   "ValveMachine_PB_Connector"(Enable := TRUE,
                           HMI_PB := "A03_HMI".MB3.Button.A0301.P3.Fermi,
                           LB_PB_Rest := FALSE,
                           LB_PB_Work := FALSE,
                           LB_PB_StartStop := FALSE,
                           Other_PB := "A03_HMI".MB3.Button.PB_Empty.Valve,
                           PB => "A0301_Fermi_P3".Fermi[1].DataIn.PB);
END_REGION

REGION Network 4 (SCL): DataIn - Fermi [1..6]
   // TRASFERIMENTO STATO PULSANTI - Comando manuale diretto 
   "A0301_Fermi_P3".Fermi[6].DataIn.PB.Rest := "A0301_Fermi_P3".Fermi[5].DataIn.PB.Rest := "A0301_Fermi_P3".Fermi[4].DataIn.PB.Rest :=
   "A0301_Fermi_P3".Fermi[3].DataIn.PB.Rest := "A0301_Fermi_P3".Fermi[2].DataIn.PB.Rest := "A0301_Fermi_P3".Fermi[1].DataIn.PB.Rest;

   "A0301_Fermi_P3".Fermi[6].DataIn.PB.Work := "A0301_Fermi_P3".Fermi[5].DataIn.PB.Work := "A0301_Fermi_P3".Fermi[4].DataIn.PB.Work :=
   "A0301_Fermi_P3".Fermi[3].DataIn.PB.Work := "A0301_Fermi_P3".Fermi[2].DataIn.PB.Work := "A0301_Fermi_P3".Fermi[1].DataIn.PB.Work;
END_REGION

REGION Network 5: << RICHIAMO STAZIONE 3 - FERMI P3 >>
   RUNG wire#powerrail
      "A0301_Fermi_P3"(AreaInterface := "Area03".AreaInterface, ZSI := "F_DB".ZSI_Zone21, DSI := "F_DB".DSI_V_Air_A0301_A0302, DataIn :=, CIn :=, Config := "PrjConfig_A03".A0301.Fermi_P3, MachineInterface =>, COut =>)
   END_RUNG
   // the same network as SCL:
   "A0301_Fermi_P3"(AreaInterface := "Area03".AreaInterface,   // "A0301_Fermi_P3_FB"
                    ZSI := "F_DB".ZSI_Zone21,
                    DSI := "F_DB".DSI_V_Air_A0301_A0302,
                    Config := "PrjConfig_A03".A0301.Fermi_P3);
END_REGION

REGION Network 6 (SCL): << TRASFERIMENTO stati DataOut >>
    REGION COMANDO DELLE USCITE FERMI P3

       // Fermi blocco prodotto Stazione P3 - RIPOSO

        "A0301_CinghiaTrasporto_1.2_V_Rest_1" := "A0301_Fermi_P3".Fermi[1].DataOut.RestSolenoid;
        "A0301_CinghiaTrasporto_2.2_V_Rest_1" := "A0301_Fermi_P3".Fermi[2].DataOut.RestSolenoid;
        "A0301_CinghiaTrasporto_3.2_V_Rest_1" := "A0301_Fermi_P3".Fermi[3].DataOut.RestSolenoid;
        "A0301_CinghiaTrasporto_4.2_V_Rest_1" := "A0301_Fermi_P3".Fermi[4].DataOut.RestSolenoid;
        "A0301_CinghiaTrasporto_5.2_V_Rest_1" := "A0301_Fermi_P3".Fermi[5].DataOut.RestSolenoid;
        "A0301_CinghiaTrasporto_6.2_V_Rest_1" := "A0301_Fermi_P3".Fermi[6].DataOut.RestSolenoid;

       // Fermi blocco prodotto Stazione P3 - LAVORO
       // 
        "A0301_CinghiaTrasporto_1.2_V_Work_2" := "A0301_Fermi_P3".Fermi[1].DataOut.WorkSolenoid;
        "A0301_CinghiaTrasporto_2.2_V_Work_2" := "A0301_Fermi_P3".Fermi[2].DataOut.WorkSolenoid;
        "A0301_CinghiaTrasporto_3.2_V_Work_2" := "A0301_Fermi_P3".Fermi[3].DataOut.WorkSolenoid;
        "A0301_CinghiaTrasporto_4.2_V_Work_2" := "A0301_Fermi_P3".Fermi[4].DataOut.WorkSolenoid;
        "A0301_CinghiaTrasporto_5.2_V_Work_2" := "A0301_Fermi_P3".Fermi[5].DataOut.WorkSolenoid;
        "A0301_CinghiaTrasporto_6.2_V_Work_2" := "A0301_Fermi_P3".Fermi[6].DataOut.WorkSolenoid;

   END_REGION ;
END_REGION
END_FUNCTION

FUNCTION_BLOCK "A0301_Fermi_P3_FB"   // FB65, LAD
// stored: MemoryReserve 100, SetENOAutomatically false
   VAR_INPUT
      AreaInterface : "AreaInterface";
      ZSI : "udt_ZoneSafetyInterface";
      DSI : "udt_DeviceSafetyInterface";
      DataIn : Struct
         OP_Rest_PB : Bool;
         OP_Work_PB : Bool;
      END_STRUCT;
      CIn : Struct
         Manager : "ValveMachine_Manager";
         SemiAut : Bool;
         P2 : Struct
            Fermi : "ValveMachine_COut";
            Sollevatore : "ValveMachine_COut";
         END_STRUCT;
         Trasporto : "SpeedMachine_COut";
      END_STRUCT;
      Config : Struct
         Fermi : Array[1..6] of "ValveMachine_Config";
         DelayMissingCondition : Time := T#3s;
      END_STRUCT;
   END_VAR
   VAR_OUTPUT
      MachineInterface : "MachineInterface";
      COut : Struct
         Fermi : "ValveMachine_COut";
      END_STRUCT;
   END_VAR
   VAR
      Alarm : Struct
         Fermi : Array[1..6] of "ValveAlr";
      END_STRUCT;
      Warning : Struct
         OP_REST_MissingCnd : Bool;   // Mancanza comando arresto
         OP_WORK_MissingCnd : Bool;   // Mancanza consenso lavoro
         Fermi : Array[1..6] of "ValveMachine_Wng";
      END_STRUCT;
      HMI : Struct
         Selection : Array[1..6] of Bool;   // 0=Disable / 1=Enable Pin
         FermiSts { S7_SetPoint := 'True'} : "UDT_HMI-Sts_ValvePosA0301";
         B_ResetShiftDone : Bool;
      END_STRUCT;
      Sts : Struct
         Fermi_AlarmPresence : Bool;
         OP_CanMoveFreely : Bool;
         OP_Rest_Cnd : Bool;
         Op_Work_Cnd : Bool;
      END_STRUCT;
      Ctrl : Struct
         OP_Rest_Man : Bool;
         OP_Work_Man : Bool;
         OP_Rest_Aut : Bool;
         OP_Work_Aut : Bool;
         OP_Rest : Bool;
         OP_Work : Bool;
      END_STRUCT;
      Fermi { S7_SetPoint := 'True'} : Array[1..6] of "ValveMachine_FB";
      AUX : Struct
         OP_Rest_PB : Bool;
         OP_Work_PB : Bool;
      END_STRUCT;
      TON_OP_REST_MissingCnd { S7_SetPoint := 'True'} : TON_TIME;
      TON_OP_WORK_MissingCnd { S7_SetPoint := 'True'} : TON_TIME;
   END_VAR
   VAR_TEMP
      PE : Struct
         OP_Rest_PB : Bool;
         OP_Work_PB : Bool;
      END_STRUCT;
      Ctrl_OLD : Struct
         CheckCndz1_ToRibalta : Bool;   // Check conditions to P3
         CheckCndz2_ToRibalta : Bool;
      END_STRUCT;
   END_VAR
   VAR_TEMP   // added for the SCL form of the ladder/FBD networks
      _w1 : Bool;
      _w2 : Bool;
      _w3 : Bool;
      _w4 : Bool;
      _w5 : Bool;
   END_VAR
BEGIN

REGION Network 2: Operazione può muoversi liberamente perchè non sposta nessun BEAM o SEMI-GUSCIO
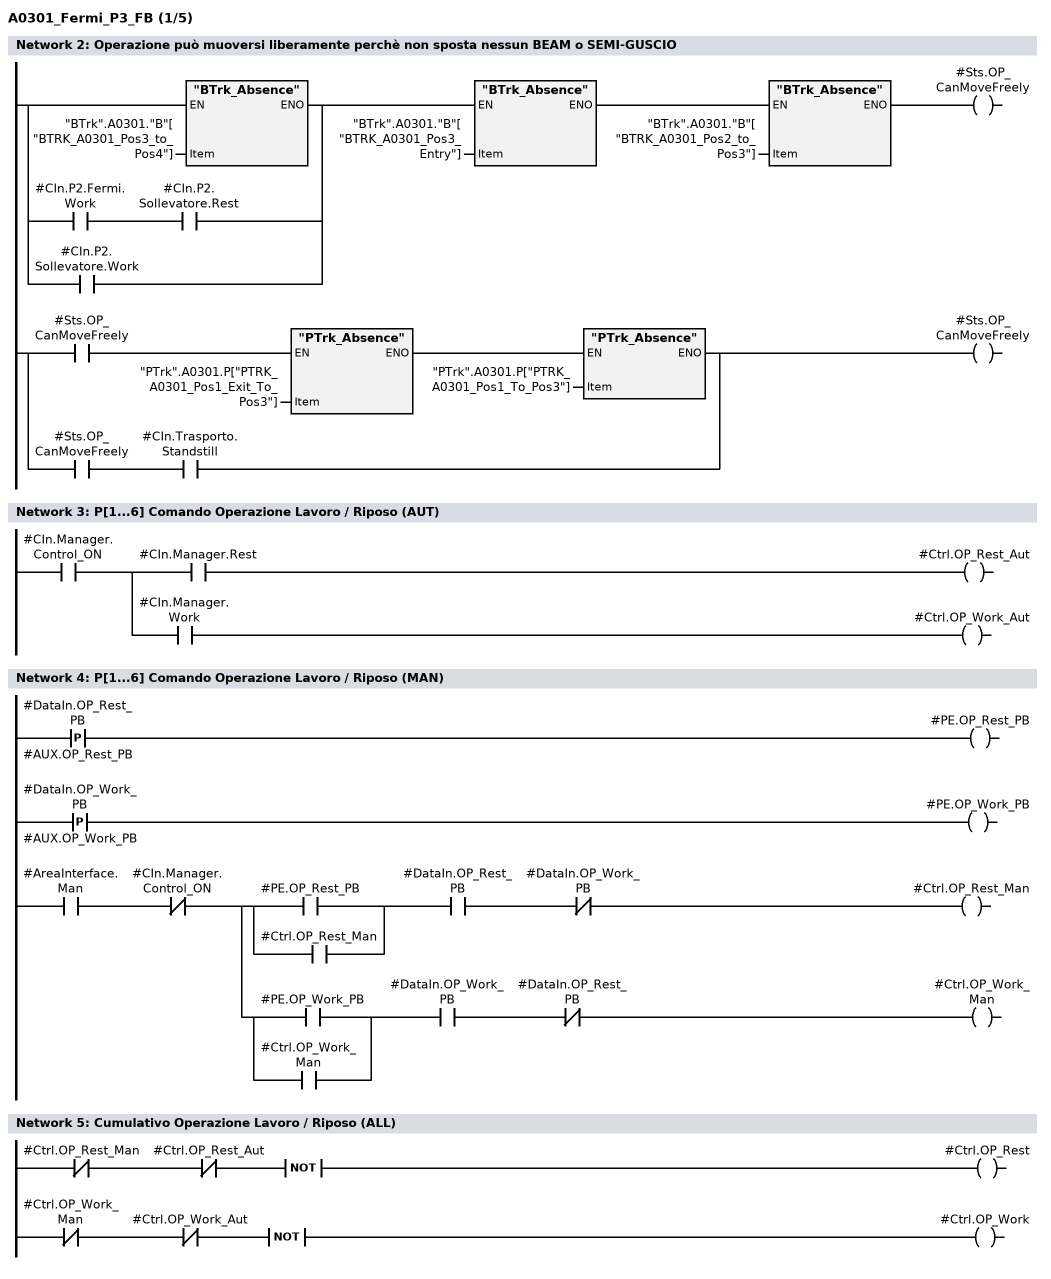
   RUNG wire#powerrail
      "BTrk_Absence"(Item := "BTrk".A0301."B"["BTRK_A0301_Pos3_to_Pos4"])
      wire#w1
      "BTrk_Absence"(Item := "BTrk".A0301."B"["BTRK_A0301_Pos3_Entry"])
      "BTrk_Absence"(Item := "BTrk".A0301."B"["BTRK_A0301_Pos2_to_Pos3"])
      Coil( #Sts.OP_CanMoveFreely )
   END_RUNG
   RUNG wire#powerrail
      Contact( #CIn.P2.Fermi.Work )
      Contact( #CIn.P2.Sollevatore.Rest )
   END_RUNG wire#w1
   RUNG wire#powerrail
      Contact( #CIn.P2.Sollevatore.Work )
   END_RUNG wire#w1
   RUNG wire#powerrail
      Contact( #Sts.OP_CanMoveFreely )
      "PTrk_Absence"(Item := "PTrk".A0301.P["PTRK_A0301_Pos1_Exit_To_Pos3"])
      "PTrk_Absence"(Item := "PTrk".A0301.P["PTRK_A0301_Pos1_To_Pos3"])
      wire#w2
      Coil( #Sts.OP_CanMoveFreely )
   END_RUNG
   RUNG wire#powerrail
      Contact( #Sts.OP_CanMoveFreely )
      Contact( #CIn.Trasporto.Standstill )
   END_RUNG wire#w2
   // the same network as SCL:
   "BTrk_Absence"(Item := "BTrk".A0301."B"["BTRK_A0301_Pos3_to_Pos4"], ENO => #_w1);
   "BTrk_Absence"(EN := #_w1 OR (#CIn.P2.Fermi.Work AND #CIn.P2.Sollevatore.Rest) OR #CIn.P2.Sollevatore.Work,
                  Item := "BTrk".A0301."B"["BTRK_A0301_Pos3_Entry"],
                  ENO => #_w2);
   "BTrk_Absence"(EN := #_w2, Item := "BTrk".A0301."B"["BTRK_A0301_Pos2_to_Pos3"], ENO => #_w3);
   #Sts.OP_CanMoveFreely := #_w3;
   "PTrk_Absence"(EN := #Sts.OP_CanMoveFreely,
                  Item := "PTrk".A0301.P["PTRK_A0301_Pos1_Exit_To_Pos3"],
                  ENO => #_w4);
   "PTrk_Absence"(EN := #_w4, Item := "PTrk".A0301.P["PTRK_A0301_Pos1_To_Pos3"], ENO => #_w5);
   #Sts.OP_CanMoveFreely := #_w5 OR (#Sts.OP_CanMoveFreely AND #CIn.Trasporto.Standstill);
END_REGION

REGION Network 3: P[1...6] Comando Operazione Lavoro / Riposo (AUT)
   RUNG wire#powerrail
      Contact( #CIn.Manager.Control_ON )
      wire#w1
      Contact( #CIn.Manager.Rest )
      Coil( #Ctrl.OP_Rest_Aut )
   END_RUNG
   RUNG wire#w1
      Contact( #CIn.Manager.Work )
      Coil( #Ctrl.OP_Work_Aut )
   END_RUNG
   // the same network as SCL:
   #Ctrl.OP_Rest_Aut := #CIn.Manager.Control_ON AND #CIn.Manager.Rest;
   #Ctrl.OP_Work_Aut := #CIn.Manager.Control_ON AND #CIn.Manager.Work;
END_REGION

REGION Network 4: P[1...6] Comando Operazione Lavoro / Riposo (MAN)
   RUNG wire#powerrail
      P_Contact(operand := #DataIn.OP_Rest_PB, bit := #AUX.OP_Rest_PB)
      Coil( #PE.OP_Rest_PB )
   END_RUNG
   RUNG wire#powerrail
      P_Contact(operand := #DataIn.OP_Work_PB, bit := #AUX.OP_Work_PB)
      Coil( #PE.OP_Work_PB )
   END_RUNG
   RUNG wire#powerrail
      Contact( #AreaInterface.Man )
      I_Contact( #CIn.Manager.Control_ON )
      wire#w1
      Contact( #PE.OP_Rest_PB )
      wire#w2
      Contact( #DataIn.OP_Rest_PB )
      I_Contact( #DataIn.OP_Work_PB )
      Coil( #Ctrl.OP_Rest_Man )
   END_RUNG
   RUNG wire#w1
      Contact( #Ctrl.OP_Rest_Man )
   END_RUNG wire#w2
   RUNG wire#w1
      Contact( #PE.OP_Work_PB )
      wire#w3
      Contact( #DataIn.OP_Work_PB )
      I_Contact( #DataIn.OP_Rest_PB )
      Coil( #Ctrl.OP_Work_Man )
   END_RUNG
   RUNG wire#w1
      Contact( #Ctrl.OP_Work_Man )
   END_RUNG wire#w3
   // the same network as SCL:
   #_w1 := #DataIn.OP_Rest_PB AND NOT #AUX.OP_Rest_PB;   // rising edge of #DataIn.OP_Rest_PB
   #AUX.OP_Rest_PB := #DataIn.OP_Rest_PB;
   #PE.OP_Rest_PB := #_w1;
   #_w2 := #DataIn.OP_Work_PB AND NOT #AUX.OP_Work_PB;   // rising edge of #DataIn.OP_Work_PB
   #AUX.OP_Work_PB := #DataIn.OP_Work_PB;
   #PE.OP_Work_PB := #_w2;
   #_w3 := #AreaInterface.Man AND NOT #CIn.Manager.Control_ON;
   #Ctrl.OP_Rest_Man := #_w3 AND (#PE.OP_Rest_PB OR #Ctrl.OP_Rest_Man) AND #DataIn.OP_Rest_PB AND NOT #DataIn.OP_Work_PB;
   #Ctrl.OP_Work_Man := #_w3 AND (#PE.OP_Work_PB OR #Ctrl.OP_Work_Man) AND #DataIn.OP_Work_PB AND NOT #DataIn.OP_Rest_PB;
END_REGION

REGION Network 5: Cumulativo Operazione Lavoro / Riposo (ALL)
   RUNG wire#powerrail
      I_Contact( #Ctrl.OP_Rest_Man )
      I_Contact( #Ctrl.OP_Rest_Aut )
      Not()
      Coil( #Ctrl.OP_Rest )
   END_RUNG
   RUNG wire#powerrail
      I_Contact( #Ctrl.OP_Work_Man )
      I_Contact( #Ctrl.OP_Work_Aut )
      Not()
      Coil( #Ctrl.OP_Work )
   END_RUNG
   // the same network as SCL:
   #Ctrl.OP_Rest := NOT (NOT #Ctrl.OP_Rest_Man AND NOT #Ctrl.OP_Rest_Aut);
   #Ctrl.OP_Work := NOT (NOT #Ctrl.OP_Work_Man AND NOT #Ctrl.OP_Work_Aut);
END_REGION

REGION Network 6: Condizioni movimento Operazione a Lavoro / Riposo
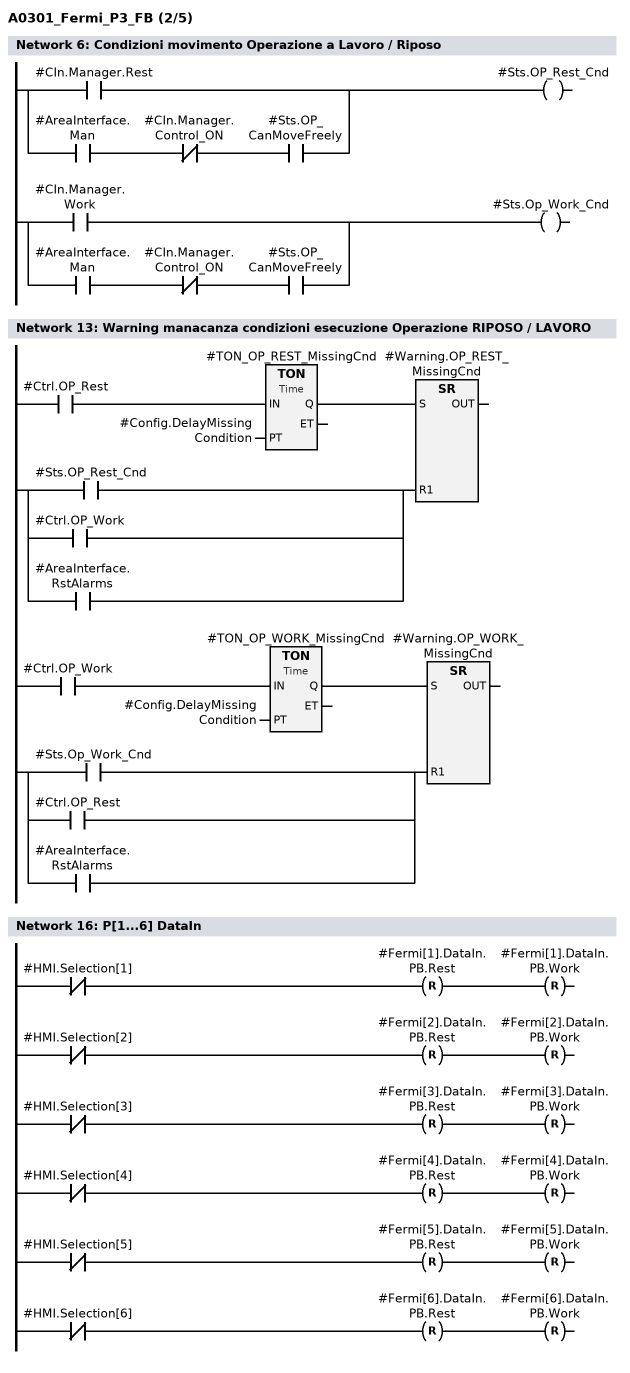
   RUNG wire#powerrail
      Contact( #CIn.Manager.Rest )
      wire#w1
      Coil( #Sts.OP_Rest_Cnd )
   END_RUNG
   RUNG wire#powerrail
      Contact( #AreaInterface.Man )
      I_Contact( #CIn.Manager.Control_ON )
      Contact( #Sts.OP_CanMoveFreely )
   END_RUNG wire#w1
   RUNG wire#powerrail
      Contact( #CIn.Manager.Work )
      wire#w2
      Coil( #Sts.Op_Work_Cnd )
   END_RUNG
   RUNG wire#powerrail
      Contact( #AreaInterface.Man )
      I_Contact( #CIn.Manager.Control_ON )
      Contact( #Sts.OP_CanMoveFreely )
   END_RUNG wire#w2
   // the same network as SCL:
   #Sts.OP_Rest_Cnd := #CIn.Manager.Rest OR (#AreaInterface.Man AND NOT #CIn.Manager.Control_ON AND #Sts.OP_CanMoveFreely);
   #Sts.Op_Work_Cnd := #CIn.Manager.Work OR (#AreaInterface.Man AND NOT #CIn.Manager.Control_ON AND #Sts.OP_CanMoveFreely);
END_REGION

REGION Network 8 (SCL): Fermi - Cin Manager (Esecuzione sequenza comandi)
   //
   #Fermi[1].Cin.Manager.Rest := FALSE;
   #Fermi[2].Cin.Manager.Rest := FALSE;
   #Fermi[3].Cin.Manager.Rest := FALSE;
   #Fermi[4].Cin.Manager.Rest := FALSE;
   #Fermi[5].Cin.Manager.Rest := FALSE;
   #Fermi[6].Cin.Manager.Rest := FALSE;

   //************************************
   #Fermi[1].Cin.Manager.Work := FALSE;
   #Fermi[2].Cin.Manager.Work := FALSE;
   #Fermi[3].Cin.Manager.Work := FALSE;
   #Fermi[4].Cin.Manager.Work := FALSE;
   #Fermi[5].Cin.Manager.Work := FALSE;
   #Fermi[6].Cin.Manager.Work := FALSE;

   //
   // CIn Manager  Control ON se ho un richiesta di comando attiva
   IF #AreaInterface.Aut OR #CIn.SemiAut THEN
       #Fermi[1].Cin.Manager.Control_ON := TRUE;
       #Fermi[2].Cin.Manager.Control_ON := TRUE;
       #Fermi[3].Cin.Manager.Control_ON := TRUE;
       #Fermi[4].Cin.Manager.Control_ON := TRUE;
       #Fermi[5].Cin.Manager.Control_ON := TRUE;
       #Fermi[6].Cin.Manager.Control_ON := TRUE;
   ELSE
       #Fermi[1].Cin.Manager.Control_ON := FALSE;
       #Fermi[2].Cin.Manager.Control_ON := FALSE;
       #Fermi[3].Cin.Manager.Control_ON := FALSE;
       #Fermi[4].Cin.Manager.Control_ON := FALSE;
       #Fermi[5].Cin.Manager.Control_ON := FALSE;
       #Fermi[6].Cin.Manager.Control_ON := FALSE;
   END_IF;

   // Comando CIn Manager Work FERMI se Sfalsatore indietro
   IF #Ctrl.OP_Work AND #Sts.Op_Work_Cnd THEN

       #Fermi[1].Cin.Manager.Work := TRUE;
       #Fermi[2].Cin.Manager.Work := TRUE;
       #Fermi[3].Cin.Manager.Work := TRUE;
       #Fermi[4].Cin.Manager.Work := TRUE;
       #Fermi[5].Cin.Manager.Work := TRUE;
       #Fermi[6].Cin.Manager.Work := TRUE;

   END_IF;

   // Comando CIn Manager Rest FERMI se Sfalsatore è basso
   IF #Ctrl.OP_Rest AND #Sts.OP_Rest_Cnd THEN

   #Fermi[1].Cin.Manager.Rest := TRUE;
   #Fermi[2].Cin.Manager.Rest := TRUE;
   #Fermi[3].Cin.Manager.Rest := TRUE;
   #Fermi[4].Cin.Manager.Rest := TRUE;
   #Fermi[5].Cin.Manager.Rest := TRUE;
   #Fermi[6].Cin.Manager.Rest := TRUE;

   END_IF;
END_REGION

REGION Network 9: <+>
END_REGION

REGION Network 10 (SCL): P[1...6] Cin Manager Comando arresto / lavoro
   //
   #Fermi[1].Cin.Manager.Rest := FALSE;
   #Fermi[2].Cin.Manager.Rest := FALSE;
   #Fermi[3].Cin.Manager.Rest := FALSE;
   #Fermi[4].Cin.Manager.Rest := FALSE;
   #Fermi[5].Cin.Manager.Rest := FALSE;
   #Fermi[6].Cin.Manager.Rest := FALSE;
   //************************************
   #Fermi[1].Cin.Manager.Work := FALSE;
   #Fermi[2].Cin.Manager.Work := FALSE;
   #Fermi[3].Cin.Manager.Work := FALSE;
   #Fermi[4].Cin.Manager.Work := FALSE;
   #Fermi[5].Cin.Manager.Work := FALSE;
   #Fermi[6].Cin.Manager.Work := FALSE;
   //
   // CIn Manager  Control ON se ho un richiesta di comando attiva
   IF #Ctrl.OP_Rest_Aut OR #Ctrl.OP_Work_Aut THEN
       #Fermi[1].Cin.Manager.Control_ON := TRUE;
       #Fermi[2].Cin.Manager.Control_ON := TRUE;
       #Fermi[3].Cin.Manager.Control_ON := TRUE;
       #Fermi[4].Cin.Manager.Control_ON := TRUE;
       #Fermi[5].Cin.Manager.Control_ON := TRUE;
       #Fermi[6].Cin.Manager.Control_ON := TRUE;
   ELSE
       #Fermi[1].Cin.Manager.Control_ON := FALSE;
       #Fermi[2].Cin.Manager.Control_ON := FALSE;
       #Fermi[3].Cin.Manager.Control_ON := FALSE;
       #Fermi[4].Cin.Manager.Control_ON := FALSE;
       #Fermi[5].Cin.Manager.Control_ON := FALSE;
       #Fermi[6].Cin.Manager.Control_ON := FALSE;
   END_IF;

   // CIn Manager Rest se ho un richiesta di comando arresto attiva
   IF #Ctrl.OP_Rest AND #Sts.OP_Rest_Cnd THEN

       #Fermi[1].Cin.Manager.Rest := TRUE;
       #Fermi[2].Cin.Manager.Rest := TRUE;
       #Fermi[3].Cin.Manager.Rest := TRUE;
       #Fermi[4].Cin.Manager.Rest := TRUE;
       #Fermi[5].Cin.Manager.Rest := TRUE;
       #Fermi[6].Cin.Manager.Rest := TRUE;

       // CIn Manager Work se ho un richiesta di comando lavoro attiva   
   ELSIF #Ctrl.OP_Work AND #Sts.Op_Work_Cnd THEN

       #Fermi[1].Cin.Manager.Work := TRUE;
       #Fermi[2].Cin.Manager.Work := TRUE;
       #Fermi[3].Cin.Manager.Work := TRUE;
       #Fermi[4].Cin.Manager.Work := TRUE;
       #Fermi[5].Cin.Manager.Work := TRUE;
       #Fermi[6].Cin.Manager.Work := TRUE;

   END_IF;
END_REGION

REGION Network 11 (SCL): P[1...6] CIn Abilitazioni Stop Manager
   //
   // CIn Manager Stop per richiesta apertura safety
   IF #CIn.Manager.EnableStopDoorOpeningReq THEN
       #Fermi[1].Cin.Manager.EnableStopDoorOpeningReq := TRUE;
       #Fermi[2].Cin.Manager.EnableStopDoorOpeningReq := TRUE;
       #Fermi[3].Cin.Manager.EnableStopDoorOpeningReq := TRUE;
       #Fermi[4].Cin.Manager.EnableStopDoorOpeningReq := TRUE;
       #Fermi[5].Cin.Manager.EnableStopDoorOpeningReq := TRUE;
       #Fermi[6].Cin.Manager.EnableStopDoorOpeningReq := TRUE;
   ELSE
       #Fermi[1].Cin.Manager.EnableStopDoorOpeningReq := FALSE;
       #Fermi[2].Cin.Manager.EnableStopDoorOpeningReq := FALSE;
       #Fermi[3].Cin.Manager.EnableStopDoorOpeningReq := FALSE;
       #Fermi[4].Cin.Manager.EnableStopDoorOpeningReq := FALSE;
       #Fermi[5].Cin.Manager.EnableStopDoorOpeningReq := FALSE;
       #Fermi[6].Cin.Manager.EnableStopDoorOpeningReq := FALSE;
   END_IF;
   // CIn Manager Stop in fase delle macchine precedenti
   IF #CIn.Manager.EnableStopInPhase THEN
       #Fermi[1].Cin.Manager.EnableStopInPhase := TRUE;
       #Fermi[2].Cin.Manager.EnableStopInPhase := TRUE;
       #Fermi[3].Cin.Manager.EnableStopInPhase := TRUE;
       #Fermi[4].Cin.Manager.EnableStopInPhase := TRUE;
       #Fermi[5].Cin.Manager.EnableStopInPhase := TRUE;
       #Fermi[6].Cin.Manager.EnableStopInPhase := TRUE;
   ELSE
       #Fermi[1].Cin.Manager.EnableStopInPhase := FALSE;
       #Fermi[2].Cin.Manager.EnableStopInPhase := FALSE;
       #Fermi[3].Cin.Manager.EnableStopInPhase := FALSE;
       #Fermi[4].Cin.Manager.EnableStopInPhase := FALSE;
       #Fermi[5].Cin.Manager.EnableStopInPhase := FALSE;
       #Fermi[6].Cin.Manager.EnableStopInPhase := FALSE;
   END_IF;

   // CIn Manager Stop programmato configurabile a piacere
   IF #CIn.Manager.EnableStopProgrammed THEN
       #Fermi[1].Cin.Manager.EnableStopProgrammed := TRUE;
       #Fermi[2].Cin.Manager.EnableStopProgrammed := TRUE;
       #Fermi[3].Cin.Manager.EnableStopProgrammed := TRUE;
       #Fermi[4].Cin.Manager.EnableStopProgrammed := TRUE;
       #Fermi[5].Cin.Manager.EnableStopProgrammed := TRUE;
       #Fermi[6].Cin.Manager.EnableStopProgrammed := TRUE;
   ELSE
       #Fermi[1].Cin.Manager.EnableStopProgrammed := FALSE;
       #Fermi[2].Cin.Manager.EnableStopProgrammed := FALSE;
       #Fermi[3].Cin.Manager.EnableStopProgrammed := FALSE;
       #Fermi[4].Cin.Manager.EnableStopProgrammed := FALSE;
       #Fermi[5].Cin.Manager.EnableStopProgrammed := FALSE;
       #Fermi[6].Cin.Manager.EnableStopProgrammed := FALSE;
   END_IF;
END_REGION

REGION Network 12: <+>
END_REGION

REGION Network 13: Warning manacanza condizioni esecuzione Operazione RIPOSO / LAVORO
   RUNG wire#powerrail
      Contact( #Ctrl.OP_Rest )
      { S7_Templates := "time_type := Time" } #TON_OP_REST_MissingCnd.TON(pt := #Config.DelayMissingCondition, et =>)
      S_SR(operand := #Warning.OP_REST_MissingCnd, r1 := wire#w1)
   END_RUNG
   RUNG wire#powerrail
      Contact( #Sts.OP_Rest_Cnd )
   END_RUNG wire#w1
   RUNG wire#powerrail
      Contact( #Ctrl.OP_Work )
   END_RUNG wire#w1
   RUNG wire#powerrail
      Contact( #AreaInterface.RstAlarms )
   END_RUNG wire#w1
   RUNG wire#powerrail
      Contact( #Ctrl.OP_Work )
      { S7_Templates := "time_type := Time" } #TON_OP_WORK_MissingCnd.TON(pt := #Config.DelayMissingCondition, et =>)
      S_SR(operand := #Warning.OP_WORK_MissingCnd, r1 := wire#w2)
   END_RUNG
   RUNG wire#powerrail
      Contact( #Sts.Op_Work_Cnd )
   END_RUNG wire#w2
   RUNG wire#powerrail
      Contact( #Ctrl.OP_Rest )
   END_RUNG wire#w2
   RUNG wire#powerrail
      Contact( #AreaInterface.RstAlarms )
   END_RUNG wire#w2
   // the same network as SCL:
   #TON_OP_REST_MissingCnd(IN := #Ctrl.OP_Rest, PT := #Config.DelayMissingCondition);   // TON
   IF #TON_OP_REST_MissingCnd.Q THEN
       #Warning.OP_REST_MissingCnd := TRUE;   // SR flip-flop
   END_IF;
   IF #Sts.OP_Rest_Cnd OR #Ctrl.OP_Work OR #AreaInterface.RstAlarms THEN
       #Warning.OP_REST_MissingCnd := FALSE;
   END_IF;
   #TON_OP_WORK_MissingCnd(IN := #Ctrl.OP_Work, PT := #Config.DelayMissingCondition);   // TON
   IF #TON_OP_WORK_MissingCnd.Q THEN
       #Warning.OP_WORK_MissingCnd := TRUE;   // SR flip-flop
   END_IF;
   IF #Sts.Op_Work_Cnd OR #Ctrl.OP_Rest OR #AreaInterface.RstAlarms THEN
       #Warning.OP_WORK_MissingCnd := FALSE;
   END_IF;
END_REGION

REGION Network 14: <+>
END_REGION

REGION Network 15: << GESTIONE FERMI >>
END_REGION

REGION Network 16: P[1...6] DataIn
   RUNG wire#powerrail
      I_Contact( #HMI.Selection[1] )
      R_Coil( #Fermi[1].DataIn.PB.Rest )
      R_Coil( #Fermi[1].DataIn.PB.Work )
   END_RUNG
   RUNG wire#powerrail
      I_Contact( #HMI.Selection[2] )
      R_Coil( #Fermi[2].DataIn.PB.Rest )
      R_Coil( #Fermi[2].DataIn.PB.Work )
   END_RUNG
   RUNG wire#powerrail
      I_Contact( #HMI.Selection[3] )
      R_Coil( #Fermi[3].DataIn.PB.Rest )
      R_Coil( #Fermi[3].DataIn.PB.Work )
   END_RUNG
   RUNG wire#powerrail
      I_Contact( #HMI.Selection[4] )
      R_Coil( #Fermi[4].DataIn.PB.Rest )
      R_Coil( #Fermi[4].DataIn.PB.Work )
   END_RUNG
   RUNG wire#powerrail
      I_Contact( #HMI.Selection[5] )
      R_Coil( #Fermi[5].DataIn.PB.Rest )
      R_Coil( #Fermi[5].DataIn.PB.Work )
   END_RUNG
   RUNG wire#powerrail
      I_Contact( #HMI.Selection[6] )
      R_Coil( #Fermi[6].DataIn.PB.Rest )
      R_Coil( #Fermi[6].DataIn.PB.Work )
   END_RUNG
   // the same network as SCL:
   IF NOT #HMI.Selection[1] THEN
       #Fermi[1].DataIn.PB.Rest := FALSE;
       #Fermi[1].DataIn.PB.Work := FALSE;
   END_IF;
   IF NOT #HMI.Selection[2] THEN
       #Fermi[2].DataIn.PB.Rest := FALSE;
       #Fermi[2].DataIn.PB.Work := FALSE;
   END_IF;
   IF NOT #HMI.Selection[3] THEN
       #Fermi[3].DataIn.PB.Rest := FALSE;
       #Fermi[3].DataIn.PB.Work := FALSE;
   END_IF;
   IF NOT #HMI.Selection[4] THEN
       #Fermi[4].DataIn.PB.Rest := FALSE;
       #Fermi[4].DataIn.PB.Work := FALSE;
   END_IF;
   IF NOT #HMI.Selection[5] THEN
       #Fermi[5].DataIn.PB.Rest := FALSE;
       #Fermi[5].DataIn.PB.Work := FALSE;
   END_IF;
   IF NOT #HMI.Selection[6] THEN
       #Fermi[6].DataIn.PB.Rest := FALSE;
       #Fermi[6].DataIn.PB.Work := FALSE;
   END_IF;
END_REGION

REGION Network 17: P[1...6] CIn External alarm
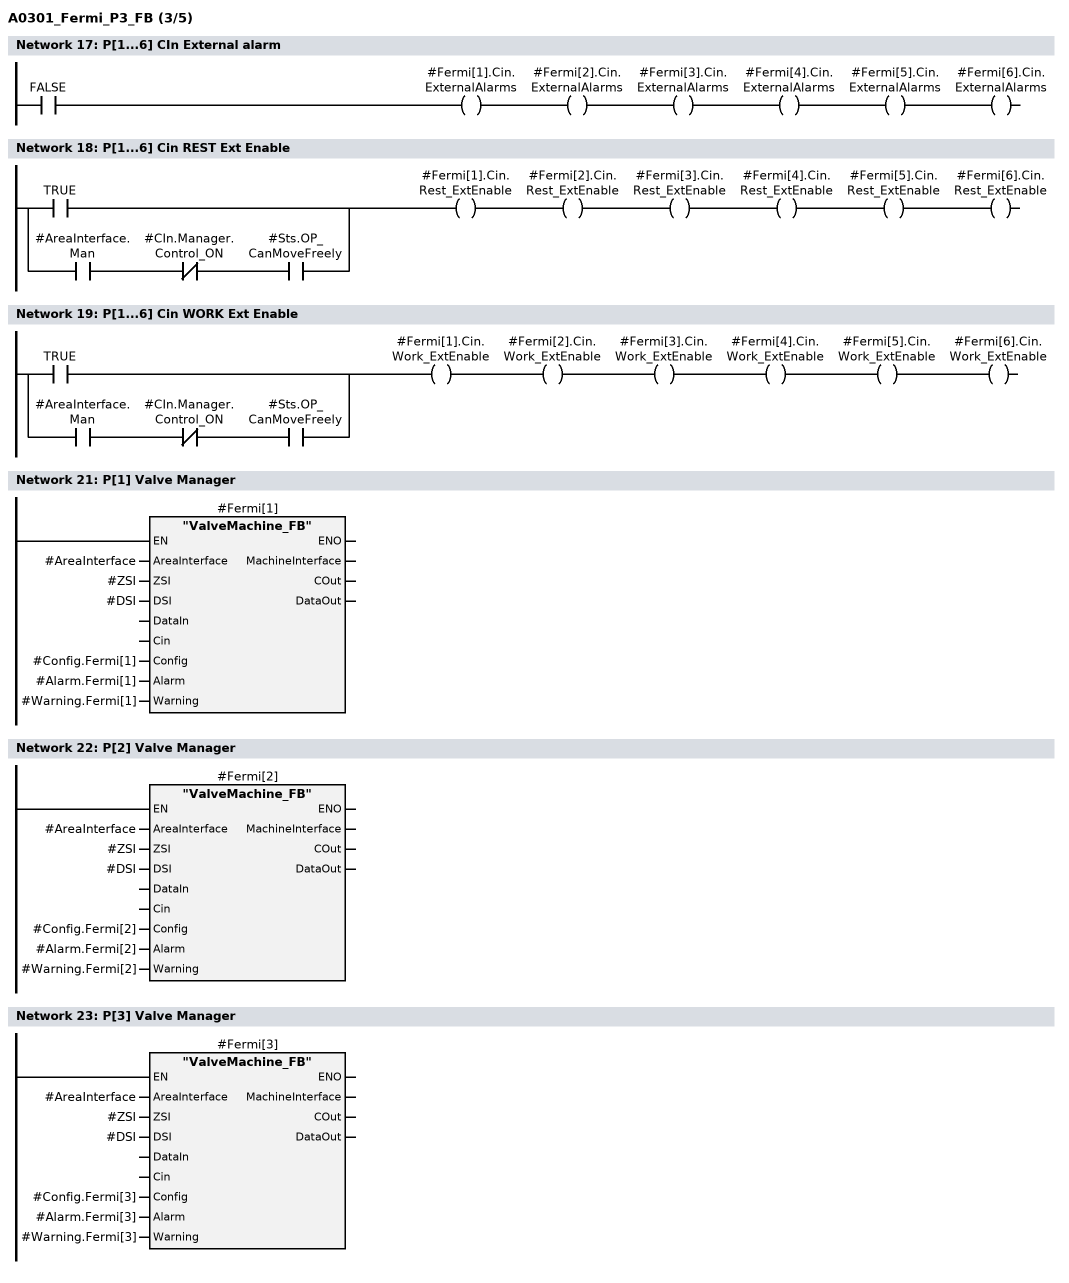
   RUNG wire#powerrail
      Contact( FALSE )
      Coil( #Fermi[1].Cin.ExternalAlarms )
      Coil( #Fermi[2].Cin.ExternalAlarms )
      Coil( #Fermi[3].Cin.ExternalAlarms )
      Coil( #Fermi[4].Cin.ExternalAlarms )
      Coil( #Fermi[5].Cin.ExternalAlarms )
      Coil( #Fermi[6].Cin.ExternalAlarms )
   END_RUNG
   // the same network as SCL:
   #Fermi[1].Cin.ExternalAlarms := FALSE;
   #Fermi[2].Cin.ExternalAlarms := FALSE;
   #Fermi[3].Cin.ExternalAlarms := FALSE;
   #Fermi[4].Cin.ExternalAlarms := FALSE;
   #Fermi[5].Cin.ExternalAlarms := FALSE;
   #Fermi[6].Cin.ExternalAlarms := FALSE;
END_REGION

REGION Network 18: P[1...6] Cin REST Ext Enable
   RUNG wire#powerrail
      Contact( TRUE )
      wire#w1
      Coil( #Fermi[1].Cin.Rest_ExtEnable )
      Coil( #Fermi[2].Cin.Rest_ExtEnable )
      Coil( #Fermi[3].Cin.Rest_ExtEnable )
      Coil( #Fermi[4].Cin.Rest_ExtEnable )
      Coil( #Fermi[5].Cin.Rest_ExtEnable )
      Coil( #Fermi[6].Cin.Rest_ExtEnable )
   END_RUNG
   RUNG wire#powerrail
      Contact( #AreaInterface.Man )
      I_Contact( #CIn.Manager.Control_ON )
      Contact( #Sts.OP_CanMoveFreely )
   END_RUNG wire#w1
   // the same network as SCL:
   #Fermi[1].Cin.Rest_ExtEnable := TRUE OR (#AreaInterface.Man AND NOT #CIn.Manager.Control_ON AND #Sts.OP_CanMoveFreely);
   #Fermi[2].Cin.Rest_ExtEnable := TRUE OR (#AreaInterface.Man AND NOT #CIn.Manager.Control_ON AND #Sts.OP_CanMoveFreely);
   #Fermi[3].Cin.Rest_ExtEnable := TRUE OR (#AreaInterface.Man AND NOT #CIn.Manager.Control_ON AND #Sts.OP_CanMoveFreely);
   #Fermi[4].Cin.Rest_ExtEnable := TRUE OR (#AreaInterface.Man AND NOT #CIn.Manager.Control_ON AND #Sts.OP_CanMoveFreely);
   #Fermi[5].Cin.Rest_ExtEnable := TRUE OR (#AreaInterface.Man AND NOT #CIn.Manager.Control_ON AND #Sts.OP_CanMoveFreely);
   #Fermi[6].Cin.Rest_ExtEnable := TRUE OR (#AreaInterface.Man AND NOT #CIn.Manager.Control_ON AND #Sts.OP_CanMoveFreely);
END_REGION

REGION Network 19: P[1...6] Cin WORK Ext Enable
   RUNG wire#powerrail
      Contact( TRUE )
      wire#w1
      Coil( #Fermi[1].Cin.Work_ExtEnable )
      Coil( #Fermi[2].Cin.Work_ExtEnable )
      Coil( #Fermi[3].Cin.Work_ExtEnable )
      Coil( #Fermi[4].Cin.Work_ExtEnable )
      Coil( #Fermi[5].Cin.Work_ExtEnable )
      Coil( #Fermi[6].Cin.Work_ExtEnable )
   END_RUNG
   RUNG wire#powerrail
      Contact( #AreaInterface.Man )
      I_Contact( #CIn.Manager.Control_ON )
      Contact( #Sts.OP_CanMoveFreely )
   END_RUNG wire#w1
   // the same network as SCL:
   #Fermi[1].Cin.Work_ExtEnable := TRUE OR (#AreaInterface.Man AND NOT #CIn.Manager.Control_ON AND #Sts.OP_CanMoveFreely);
   #Fermi[2].Cin.Work_ExtEnable := TRUE OR (#AreaInterface.Man AND NOT #CIn.Manager.Control_ON AND #Sts.OP_CanMoveFreely);
   #Fermi[3].Cin.Work_ExtEnable := TRUE OR (#AreaInterface.Man AND NOT #CIn.Manager.Control_ON AND #Sts.OP_CanMoveFreely);
   #Fermi[4].Cin.Work_ExtEnable := TRUE OR (#AreaInterface.Man AND NOT #CIn.Manager.Control_ON AND #Sts.OP_CanMoveFreely);
   #Fermi[5].Cin.Work_ExtEnable := TRUE OR (#AreaInterface.Man AND NOT #CIn.Manager.Control_ON AND #Sts.OP_CanMoveFreely);
   #Fermi[6].Cin.Work_ExtEnable := TRUE OR (#AreaInterface.Man AND NOT #CIn.Manager.Control_ON AND #Sts.OP_CanMoveFreely);
END_REGION

REGION Network 20: <+>
END_REGION

REGION Network 21: P[1] Valve Manager
   RUNG wire#powerrail
      #Fermi[1](AreaInterface := #AreaInterface, ZSI := #ZSI, DSI := #DSI, DataIn :=, Cin :=, Config := #Config.Fermi[1], Alarm := #Alarm.Fermi[1], Warning := #Warning.Fermi[1], MachineInterface =>, COut =>, DataOut =>)
   END_RUNG
   // the same network as SCL:
   #Fermi[1](AreaInterface := #AreaInterface,   // "ValveMachine_FB"
             ZSI := #ZSI,
             DSI := #DSI,
             Config := #Config.Fermi[1],
             Alarm := #Alarm.Fermi[1],
             Warning := #Warning.Fermi[1]);
END_REGION

REGION Network 22: P[2] Valve Manager
   RUNG wire#powerrail
      #Fermi[2](AreaInterface := #AreaInterface, ZSI := #ZSI, DSI := #DSI, DataIn :=, Cin :=, Config := #Config.Fermi[2], Alarm := #Alarm.Fermi[2], Warning := #Warning.Fermi[2], MachineInterface =>, COut =>, DataOut =>)
   END_RUNG
   // the same network as SCL:
   #Fermi[2](AreaInterface := #AreaInterface,   // "ValveMachine_FB"
             ZSI := #ZSI,
             DSI := #DSI,
             Config := #Config.Fermi[2],
             Alarm := #Alarm.Fermi[2],
             Warning := #Warning.Fermi[2]);
END_REGION

REGION Network 23: P[3] Valve Manager
   RUNG wire#powerrail
      #Fermi[3](AreaInterface := #AreaInterface, ZSI := #ZSI, DSI := #DSI, DataIn :=, Cin :=, Config := #Config.Fermi[3], Alarm := #Alarm.Fermi[3], Warning := #Warning.Fermi[3], MachineInterface =>, COut =>, DataOut =>)
   END_RUNG
   // the same network as SCL:
   #Fermi[3](AreaInterface := #AreaInterface,   // "ValveMachine_FB"
             ZSI := #ZSI,
             DSI := #DSI,
             Config := #Config.Fermi[3],
             Alarm := #Alarm.Fermi[3],
             Warning := #Warning.Fermi[3]);
END_REGION

REGION Network 24: P[4] Valve Manager
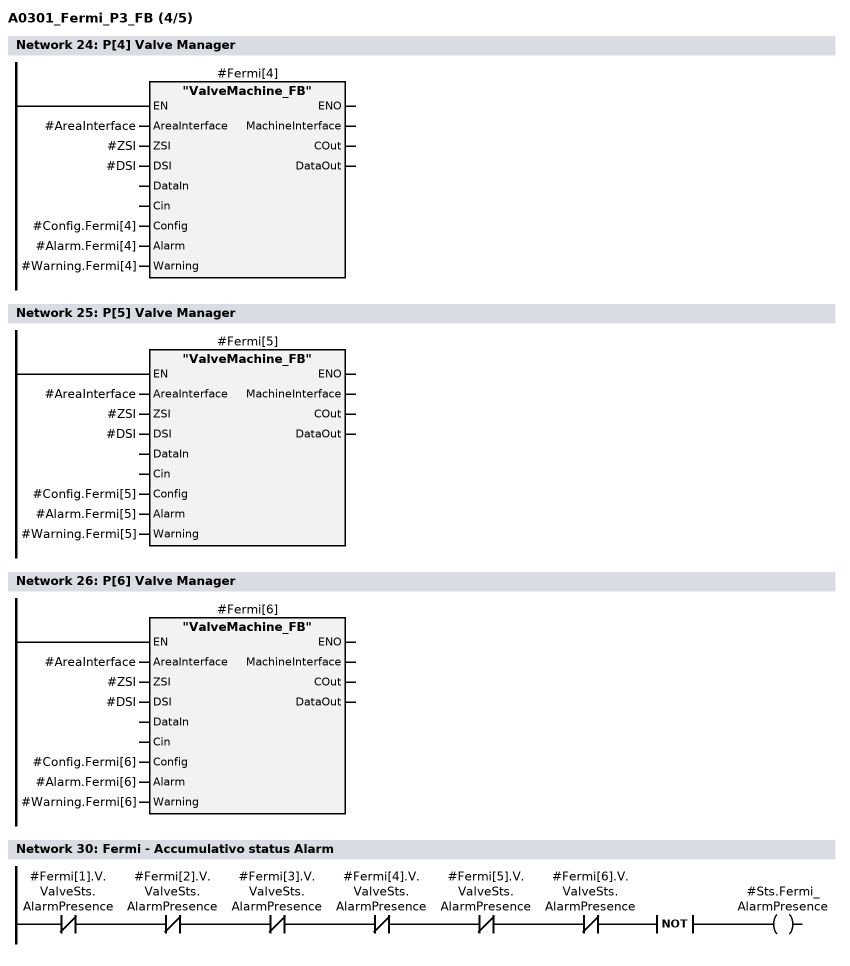
   RUNG wire#powerrail
      #Fermi[4](AreaInterface := #AreaInterface, ZSI := #ZSI, DSI := #DSI, DataIn :=, Cin :=, Config := #Config.Fermi[4], Alarm := #Alarm.Fermi[4], Warning := #Warning.Fermi[4], MachineInterface =>, COut =>, DataOut =>)
   END_RUNG
   // the same network as SCL:
   #Fermi[4](AreaInterface := #AreaInterface,   // "ValveMachine_FB"
             ZSI := #ZSI,
             DSI := #DSI,
             Config := #Config.Fermi[4],
             Alarm := #Alarm.Fermi[4],
             Warning := #Warning.Fermi[4]);
END_REGION

REGION Network 25: P[5] Valve Manager
   RUNG wire#powerrail
      #Fermi[5](AreaInterface := #AreaInterface, ZSI := #ZSI, DSI := #DSI, DataIn :=, Cin :=, Config := #Config.Fermi[5], Alarm := #Alarm.Fermi[5], Warning := #Warning.Fermi[5], MachineInterface =>, COut =>, DataOut =>)
   END_RUNG
   // the same network as SCL:
   #Fermi[5](AreaInterface := #AreaInterface,   // "ValveMachine_FB"
             ZSI := #ZSI,
             DSI := #DSI,
             Config := #Config.Fermi[5],
             Alarm := #Alarm.Fermi[5],
             Warning := #Warning.Fermi[5]);
END_REGION

REGION Network 26: P[6] Valve Manager
   RUNG wire#powerrail
      #Fermi[6](AreaInterface := #AreaInterface, ZSI := #ZSI, DSI := #DSI, DataIn :=, Cin :=, Config := #Config.Fermi[6], Alarm := #Alarm.Fermi[6], Warning := #Warning.Fermi[6], MachineInterface =>, COut =>, DataOut =>)
   END_RUNG
   // the same network as SCL:
   #Fermi[6](AreaInterface := #AreaInterface,   // "ValveMachine_FB"
             ZSI := #ZSI,
             DSI := #DSI,
             Config := #Config.Fermi[6],
             Alarm := #Alarm.Fermi[6],
             Warning := #Warning.Fermi[6]);
END_REGION

REGION Network 27: <+>
END_REGION

REGION Network 28 (SCL): P[1...6] COut Fermi
   REGION COut STANDSTILL Fermi
       // Controllo uscita COut STANDSTILL in base allo stato di tutti i Pin
       IF  #Fermi[1].Sts.Standstill AND
           #Fermi[2].Sts.Standstill AND
           #Fermi[3].Sts.Standstill AND
           #Fermi[4].Sts.Standstill AND
           #Fermi[5].Sts.Standstill AND
           #Fermi[6].Sts.Standstill THEN
           #COut.Fermi.Standstill := TRUE;
       ELSE
           #COut.Fermi.Standstill := FALSE;
       END_IF;
   END_REGION ;


   REGION COut AT REST #Fermi
       // Controllo uscita COut AT_REST in base allo stato di tutti i Pin
       IF  #Fermi[1].COut.Rest OR #Fermi[1].DataIn.Rest_Ls[1] AND
           #Fermi[2].COut.Rest OR #Fermi[2].DataIn.Rest_Ls[1] AND
           #Fermi[3].COut.Rest OR #Fermi[3].DataIn.Rest_Ls[1] AND
           #Fermi[4].COut.Rest OR #Fermi[4].DataIn.Rest_Ls[1] AND
           #Fermi[5].COut.Rest OR #Fermi[5].DataIn.Rest_Ls[1] AND
           #Fermi[6].COut.Rest OR #Fermi[6].DataIn.Rest_Ls[1] THEN
           #COut.Fermi.Rest := 1;
       ELSE
           #COut.Fermi.Rest := 0;
       END_IF;
   END_REGION ;

   REGION COut AT WORK Fermi
       // Controllo uscita COut AT_WORK in base allo stato di tutti i Pin
       IF #Fermi[1].COut.Work AND
           #Fermi[2].COut.Work AND
           #Fermi[3].COut.Work AND
           #Fermi[4].COut.Work AND
           #Fermi[5].COut.Work AND
           #Fermi[6].COut.Work THEN
           #COut.Fermi.Work := 1;
       ELSE
           #COut.Fermi.Work := 0;
       END_IF;
   END_REGION ;
END_REGION

REGION Network 30: Fermi - Accumulativo status Alarm
   RUNG wire#powerrail
      I_Contact( #Fermi[1].V.ValveSts.AlarmPresence )
      I_Contact( #Fermi[2].V.ValveSts.AlarmPresence )
      I_Contact( #Fermi[3].V.ValveSts.AlarmPresence )
      I_Contact( #Fermi[4].V.ValveSts.AlarmPresence )
      I_Contact( #Fermi[5].V.ValveSts.AlarmPresence )
      I_Contact( #Fermi[6].V.ValveSts.AlarmPresence )
      Not()
      Coil( #Sts.Fermi_AlarmPresence )
   END_RUNG
   // the same network as SCL:
   #Sts.Fermi_AlarmPresence := NOT (NOT #Fermi[1].V.ValveSts.AlarmPresence AND NOT #Fermi[2].V.ValveSts.AlarmPresence AND NOT #Fermi[3].V.ValveSts.AlarmPresence AND NOT #Fermi[4].V.ValveSts.AlarmPresence AND NOT #Fermi[5].V.ValveSts.AlarmPresence AND NOT #Fermi[6].V.ValveSts.AlarmPresence);
END_REGION

REGION Network 31 (SCL): HMI STATUS - Postazione
   // Area dati appoggio per HMI
   // FERMI POS.3
   #HMI.FermiSts.Standstill := #COut.Fermi.Standstill;
   #HMI.FermiSts.Rest := #COut.Fermi.Rest;
   #HMI.FermiSts.Work := #COut.Fermi.Work;
   #HMI.FermiSts.AlarmPresence := #Sts.Fermi_AlarmPresence;
END_REGION

REGION Network 33: << MAIN MACHINE STATUS >>
END_REGION

REGION Network 34: Machine interface
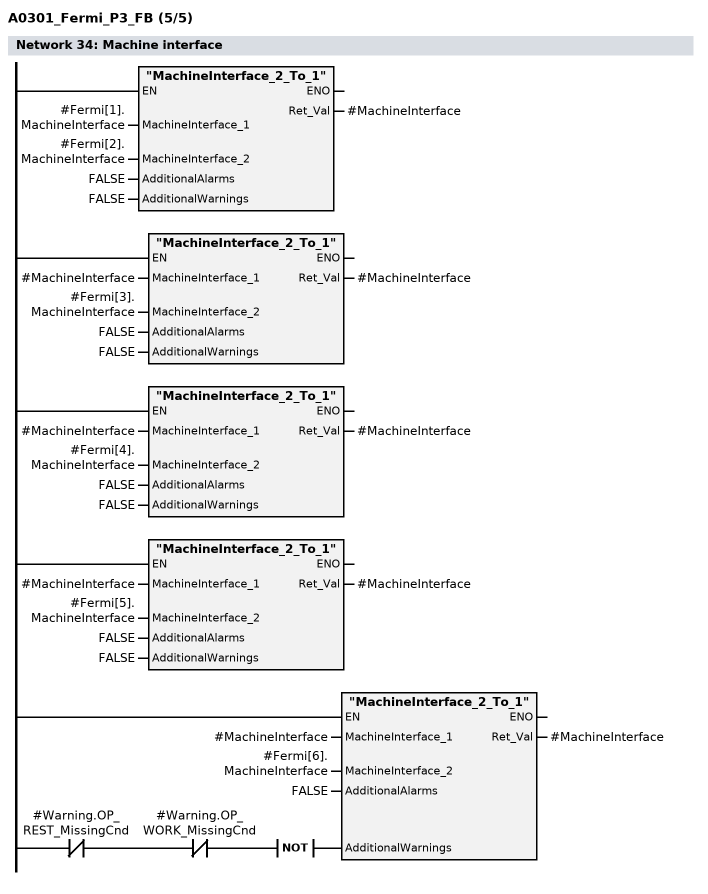
   RUNG wire#powerrail
      "MachineInterface_2_To_1"(MachineInterface_1 := #Fermi[1].MachineInterface, MachineInterface_2 := #Fermi[2].MachineInterface, AdditionalAlarms := FALSE, AdditionalWarnings := FALSE, Ret_Val => #MachineInterface)
   END_RUNG
   RUNG wire#powerrail
      "MachineInterface_2_To_1"(MachineInterface_1 := #MachineInterface, MachineInterface_2 := #Fermi[3].MachineInterface, AdditionalAlarms := FALSE, AdditionalWarnings := FALSE, Ret_Val => #MachineInterface)
   END_RUNG
   RUNG wire#powerrail
      "MachineInterface_2_To_1"(MachineInterface_1 := #MachineInterface, MachineInterface_2 := #Fermi[4].MachineInterface, AdditionalAlarms := FALSE, AdditionalWarnings := FALSE, Ret_Val => #MachineInterface)
   END_RUNG
   RUNG wire#powerrail
      "MachineInterface_2_To_1"(MachineInterface_1 := #MachineInterface, MachineInterface_2 := #Fermi[5].MachineInterface, AdditionalAlarms := FALSE, AdditionalWarnings := FALSE, Ret_Val => #MachineInterface)
   END_RUNG
   RUNG wire#powerrail
      "MachineInterface_2_To_1"(AdditionalWarnings := wire#w1, MachineInterface_1 := #MachineInterface, MachineInterface_2 := #Fermi[6].MachineInterface, AdditionalAlarms := FALSE, Ret_Val => #MachineInterface)
   END_RUNG
   RUNG wire#powerrail
      I_Contact( #Warning.OP_REST_MissingCnd )
      I_Contact( #Warning.OP_WORK_MissingCnd )
      Not()
   END_RUNG wire#w1
   // the same network as SCL:
   #MachineInterface := "MachineInterface_2_To_1"(MachineInterface_1 := #Fermi[1].MachineInterface,
                           MachineInterface_2 := #Fermi[2].MachineInterface,
                           AdditionalAlarms := FALSE,
                           AdditionalWarnings := FALSE);
   #MachineInterface := "MachineInterface_2_To_1"(MachineInterface_1 := #MachineInterface,
                           MachineInterface_2 := #Fermi[3].MachineInterface,
                           AdditionalAlarms := FALSE,
                           AdditionalWarnings := FALSE);
   #MachineInterface := "MachineInterface_2_To_1"(MachineInterface_1 := #MachineInterface,
                           MachineInterface_2 := #Fermi[4].MachineInterface,
                           AdditionalAlarms := FALSE,
                           AdditionalWarnings := FALSE);
   #MachineInterface := "MachineInterface_2_To_1"(MachineInterface_1 := #MachineInterface,
                           MachineInterface_2 := #Fermi[5].MachineInterface,
                           AdditionalAlarms := FALSE,
                           AdditionalWarnings := FALSE);
   #MachineInterface := "MachineInterface_2_To_1"(MachineInterface_1 := #MachineInterface,
                           MachineInterface_2 := #Fermi[6].MachineInterface,
                           AdditionalAlarms := FALSE,
                           AdditionalWarnings := NOT (NOT #Warning.OP_REST_MissingCnd AND NOT #Warning.OP_WORK_MissingCnd));
END_REGION
END_FUNCTION_BLOCK

FUNCTION "A0301_Ribaltatore_CALL" : Void   // FC134, LAD
// stored: SetENOAutomatically false
   VAR CONSTANT
      MinimumPos : Real := 0.0;
      MaximumPos : Real := 1000.0;
      MISSING : Int;
   END_VAR
BEGIN

REGION Network 1 (SCL): << TRASFERIMENTO stati CIn del blocco >>
   // SOSTITUIRE SYS BYPASS CON INGRESSI DIGITALI
   // TRASFERIMENTO COMANDI CIn MANAGER
   "A0301_Ribaltatore".CIn.Manager.Ax := "A0301_Manager".COut.Ribaltatore.Ax;
   "A0301_Ribaltatore".CIn.Manager.Solleva := "A0301_Manager".COut.Ribaltatore.Solleva;
   //
   "A0301_Ribaltatore".CIn.SemiAut_PB := "A0301_Manager".DataIn.SemiAut_Pb;


   REGION TRASFERIMENTO DataIn DIGITAL INPUT dei LIMIT SWITCH

       "A0301_Ribaltatore".Ax.CIn.PositionLimits.EnableMin := 1;
       "A0301_Ribaltatore".Ax.CIn.PositionLimits.EnableMax := 1;

       // Limiti di Posizione Minima & Massima (IMPOSTARE LE COSTANTI DOPO LA PROVA MANUALE)
       "A0301_Ribaltatore".Ax.CIn.PositionLimits.PosMin := #MinimumPos;
       "A0301_Ribaltatore".Ax.CIn.PositionLimits.PosMax := #MaximumPos;
   END_REGION ;

   REGION TRASFERIMENTO REQ. DI POSIZIONE E STATI
       "A0301_Ribaltatore".CIn.Ax_Req := "A0301_Manager".COut.Ribaltatore.Ax_Req;
   END_REGION ;
END_REGION

REGION Network 2 (SCL): << TRASFERIMENTO stati DataIn >>
   REGION TRASFERIMENTO #DataIn STATI BUTTON RIBALTATORE
       // PB RIBALTATORE
       "A0301_Ribaltatore".Ax.DataIn.PB.Bwd_Minus := "A03_HMI".MB3.Button.A0301.Ribaltatore.Rotazione.Bwd_Minus;
       "A0301_Ribaltatore".Ax.DataIn.PB.Fwd_Plus := "A03_HMI".MB3.Button.A0301.Ribaltatore.Rotazione.Fwd_Plus;
       "A0301_Ribaltatore".Ax.DataIn.PB.MoveToPos := "A03_HMI".MB3.Button.A0301.Ribaltatore.Rotazione.MoveToPos;


   END_REGION ;

   //SOLLEVATORE RIBALTATORE - Stato dei sensori Ls
   // EV SOLLEVA RIBALTATORE
   "A0301_Ribaltatore".Solleva_Rib[1].DataIn.Rest_Ls[1] := "A0301_CinghiaTrasporto_1.1_Ls_Rest_1";
   "A0301_Ribaltatore".Solleva_Rib[2].DataIn.Rest_Ls[1] := "A0301_CinghiaTrasporto_2.1_Ls_Rest_1";
   "A0301_Ribaltatore".Solleva_Rib[3].DataIn.Rest_Ls[1] := "A0301_CinghiaTrasporto_3.1_Ls_Rest_1";
   "A0301_Ribaltatore".Solleva_Rib[4].DataIn.Rest_Ls[1] := "A0301_CinghiaTrasporto_4.1_Ls_Rest_1";
   "A0301_Ribaltatore".Solleva_Rib[5].DataIn.Rest_Ls[1] := "A0301_CinghiaTrasporto_5.1_Ls_Rest_1";
   "A0301_Ribaltatore".Solleva_Rib[6].DataIn.Rest_Ls[1] := "A0301_CinghiaTrasporto_6.1_Ls_Rest_1";
   //
   "A0301_Ribaltatore".Solleva_Rib[1].DataIn.Work_Ls[1] := "A0301_CinghiaTrasporto_1.1_Ls_Work_2";
   "A0301_Ribaltatore".Solleva_Rib[2].DataIn.Work_Ls[1] := "A0301_CinghiaTrasporto_2.1_Ls_Work_2";
   "A0301_Ribaltatore".Solleva_Rib[3].DataIn.Work_Ls[1] := "A0301_CinghiaTrasporto_3.1_Ls_Work_2";
   "A0301_Ribaltatore".Solleva_Rib[4].DataIn.Work_Ls[1] := "A0301_CinghiaTrasporto_4.1_Ls_Work_2";
   "A0301_Ribaltatore".Solleva_Rib[5].DataIn.Work_Ls[1] := "A0301_CinghiaTrasporto_5.1_Ls_Work_2";
   "A0301_Ribaltatore".Solleva_Rib[6].DataIn.Work_Ls[1] := "A0301_CinghiaTrasporto_6.1_Ls_Work_2";

   // RIBALTATORE - Ax    
   // Trasferimento ingressi digitali Limit Switch Bassa e Alta
   "A0301_Ribaltatore".Ax.DataIn.LS_Minus :=  "A0301_Ribaltatore_Ls_Minimo";
   "A0301_Ribaltatore".Ax.DataIn.LS_Plus := "Sys".ByPass;
   //"A0301_Ribaltatore_Ls_Massimo";
   //
END_REGION

REGION Network 3: DataIn - Solleva Ribalta
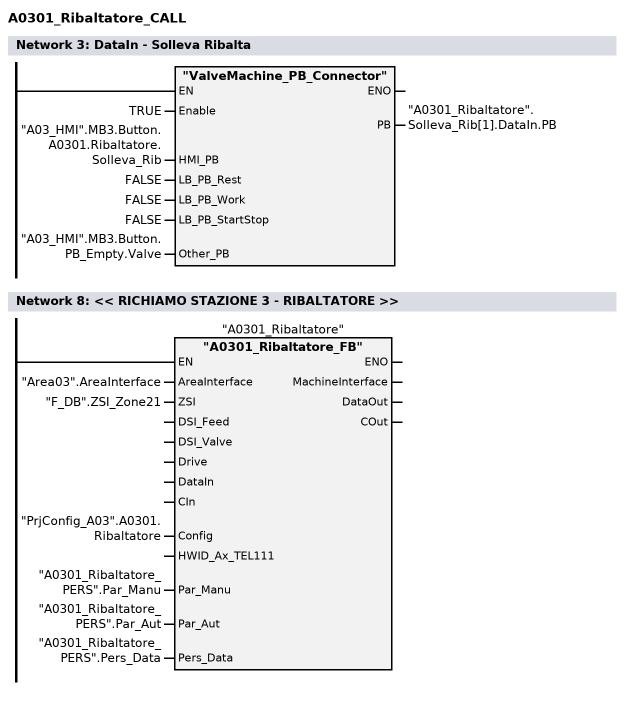
   RUNG wire#powerrail
      "ValveMachine_PB_Connector"(Enable := TRUE, HMI_PB := "A03_HMI".MB3.Button.A0301.Ribaltatore.Solleva_Rib, LB_PB_Rest := FALSE, LB_PB_Work := FALSE, LB_PB_StartStop := FALSE, Other_PB := "A03_HMI".MB3.Button.PB_Empty.Valve, PB => "A0301_Ribaltatore".Solleva_Rib[1].DataIn.PB)
   END_RUNG
   // the same network as SCL:
   "ValveMachine_PB_Connector"(Enable := TRUE,
                           HMI_PB := "A03_HMI".MB3.Button.A0301.Ribaltatore.Solleva_Rib,
                           LB_PB_Rest := FALSE,
                           LB_PB_Work := FALSE,
                           LB_PB_StartStop := FALSE,
                           Other_PB := "A03_HMI".MB3.Button.PB_Empty.Valve,
                           PB => "A0301_Ribaltatore".Solleva_Rib[1].DataIn.PB);
END_REGION

REGION Network 4 (SCL): DataIn - Fermi [1..6]
   // TRASFERIMENTO STATO PULSANTI - Comando manuale diretto 
   "A0301_Ribaltatore".Solleva_Rib[6].DataIn.PB := "A0301_Ribaltatore".Solleva_Rib[5].DataIn.PB := "A0301_Ribaltatore".Solleva_Rib[4].DataIn.PB :=
   "A0301_Ribaltatore".Solleva_Rib[3].DataIn.PB := "A0301_Ribaltatore".Solleva_Rib[2].DataIn.PB := "A0301_Ribaltatore".Solleva_Rib[1].DataIn.PB;
END_REGION

REGION Network 5 (SCL): DSI
   //
   "A0301_Ribaltatore".DSI_Feed := "F_DB".DSI_Ribaltatore;
   "A0301_Ribaltatore".DSI_Valve := "F_DB".DSI_V_Air_A0301_A0302;
END_REGION

REGION Network 6 (SCL): HW
   //
   "A0301_Ribaltatore".HWID_Ax_TEL111 := "HW_Const_Values".CU5_PN_1560A1_1_SIEMENS_telegram_111;
END_REGION

REGION Network 7 (SCL): Drive
   //
   "A0301_Ribaltatore".Drive.Infeed_ON := "Areas_ITF".AG.Infeed_Running;;
   "A0301_Ribaltatore".Drive.AccessPoint := "HW_Const_Values".CU5_PN_600A1_ModuleAccessPoint;
   "A0301_Ribaltatore".Drive.AxisID := "CU5_ID_5_1560A1_1_1560M1";
   "A0301_Ribaltatore".Drive.TokenChain := "TOKENCHAIN_CU5";
END_REGION

REGION Network 8: << RICHIAMO STAZIONE 3 - RIBALTATORE >>
   RUNG wire#powerrail
      "A0301_Ribaltatore"(AreaInterface := "Area03".AreaInterface, ZSI := "F_DB".ZSI_Zone21, DSI_Feed :=, DSI_Valve :=, Drive :=, DataIn :=, CIn :=, Config := "PrjConfig_A03".A0301.Ribaltatore, HWID_Ax_TEL111 :=, Par_Manu := "A0301_Ribaltatore_PERS".Par_Manu, Par_Aut := "A0301_Ribaltatore_PERS".Par_Aut, Pers_Data := "A0301_Ribaltatore_PERS".Pers_Data, MachineInterface =>, DataOut =>, COut =>)
   END_RUNG
   // the same network as SCL:
   "A0301_Ribaltatore"(AreaInterface := "Area03".AreaInterface,   // "A0301_Ribaltatore_FB"
                       ZSI := "F_DB".ZSI_Zone21,
                       Config := "PrjConfig_A03".A0301.Ribaltatore,
                       Par_Manu := "A0301_Ribaltatore_PERS".Par_Manu,
                       Par_Aut := "A0301_Ribaltatore_PERS".Par_Aut,
                       Pers_Data := "A0301_Ribaltatore_PERS".Pers_Data);
END_REGION

REGION Network 9 (SCL): << TRASFERIMENTO stati DataOut >>

